   // UNICODE_TO_GBK[24826] := 16#7BB0;
   // UNICODE_TO_GBK[24827] := 16#B990;
   // UNICODE_TO_GBK[24828] := 16#7BB1;
   // UNICODE_TO_GBK[24829] := 16#CFE4;
   // UNICODE_TO_GBK[24830] := 16#7BB2;
   // UNICODE_TO_GBK[24831] := 16#B991;
   // UNICODE_TO_GBK[24832] := 16#7BB3;
   // UNICODE_TO_GBK[24833] := 16#B992;
   // UNICODE_TO_GBK[24834] := 16#7BB4;
   // UNICODE_TO_GBK[24835] := 16#F3F0;
   // UNICODE_TO_GBK[24836] := 16#7BB5;
   // UNICODE_TO_GBK[24837] := 16#B993;
   // UNICODE_TO_GBK[24838] := 16#7BB6;
   // UNICODE_TO_GBK[24839] := 16#B994;
   // UNICODE_TO_GBK[24840] := 16#7BB7;
   // UNICODE_TO_GBK[24841] := 16#B995;
   // UNICODE_TO_GBK[24842] := 16#7BB8;
   // UNICODE_TO_GBK[24843] := 16#F3E7;
   // UNICODE_TO_GBK[24844] := 16#7BB9;
   // UNICODE_TO_GBK[24845] := 16#B996;
   // UNICODE_TO_GBK[24846] := 16#7BBA;
   // UNICODE_TO_GBK[24847] := 16#B997;
   // UNICODE_TO_GBK[24848] := 16#7BBB;
   // UNICODE_TO_GBK[24849] := 16#B998;
   // UNICODE_TO_GBK[24850] := 16#7BBC;
   // UNICODE_TO_GBK[24851] := 16#B999;
   // UNICODE_TO_GBK[24852] := 16#7BBD;
   // UNICODE_TO_GBK[24853] := 16#B99A;
   // UNICODE_TO_GBK[24854] := 16#7BBE;
   // UNICODE_TO_GBK[24855] := 16#B99B;
   // UNICODE_TO_GBK[24856] := 16#7BBF;
   // UNICODE_TO_GBK[24857] := 16#B99C;
   // UNICODE_TO_GBK[24858] := 16#7BC0;
   // UNICODE_TO_GBK[24859] := 16#B99D;
   // UNICODE_TO_GBK[24860] := 16#7BC1;
   // UNICODE_TO_GBK[24861] := 16#F3F2;
   // UNICODE_TO_GBK[24862] := 16#7BC2;
   // UNICODE_TO_GBK[24863] := 16#B99E;
   // UNICODE_TO_GBK[24864] := 16#7BC3;
   // UNICODE_TO_GBK[24865] := 16#B99F;
   // UNICODE_TO_GBK[24866] := 16#7BC4;
   // UNICODE_TO_GBK[24867] := 16#B9A0;
   // UNICODE_TO_GBK[24868] := 16#7BC5;
   // UNICODE_TO_GBK[24869] := 16#BA40;
   // UNICODE_TO_GBK[24870] := 16#7BC6;
   // UNICODE_TO_GBK[24871] := 16#D7AD;
   // UNICODE_TO_GBK[24872] := 16#7BC7;
   // UNICODE_TO_GBK[24873] := 16#C6AA;
   // UNICODE_TO_GBK[24874] := 16#7BC8;
   // UNICODE_TO_GBK[24875] := 16#BA41;
   // UNICODE_TO_GBK[24876] := 16#7BC9;
   // UNICODE_TO_GBK[24877] := 16#BA42;
   // UNICODE_TO_GBK[24878] := 16#7BCA;
   // UNICODE_TO_GBK[24879] := 16#BA43;
   // UNICODE_TO_GBK[24880] := 16#7BCB;
   // UNICODE_TO_GBK[24881] := 16#BA44;
   // UNICODE_TO_GBK[24882] := 16#7BCC;
   // UNICODE_TO_GBK[24883] := 16#F3F3;
   // UNICODE_TO_GBK[24884] := 16#7BCD;
   // UNICODE_TO_GBK[24885] := 16#BA45;
   // UNICODE_TO_GBK[24886] := 16#7BCE;
   // UNICODE_TO_GBK[24887] := 16#BA46;
   // UNICODE_TO_GBK[24888] := 16#7BCF;
   // UNICODE_TO_GBK[24889] := 16#BA47;
   // UNICODE_TO_GBK[24890] := 16#7BD0;
   // UNICODE_TO_GBK[24891] := 16#BA48;
   // UNICODE_TO_GBK[24892] := 16#7BD1;
   // UNICODE_TO_GBK[24893] := 16#F3F1;
   // UNICODE_TO_GBK[24894] := 16#7BD2;
   // UNICODE_TO_GBK[24895] := 16#BA49;
   // UNICODE_TO_GBK[24896] := 16#7BD3;
   // UNICODE_TO_GBK[24897] := 16#C2A8;
   // UNICODE_TO_GBK[24898] := 16#7BD4;
   // UNICODE_TO_GBK[24899] := 16#BA4A;
   // UNICODE_TO_GBK[24900] := 16#7BD5;
   // UNICODE_TO_GBK[24901] := 16#BA4B;
   // UNICODE_TO_GBK[24902] := 16#7BD6;
   // UNICODE_TO_GBK[24903] := 16#BA4C;
   // UNICODE_TO_GBK[24904] := 16#7BD7;
   // UNICODE_TO_GBK[24905] := 16#BA4D;
   // UNICODE_TO_GBK[24906] := 16#7BD8;
   // UNICODE_TO_GBK[24907] := 16#BA4E;
   // UNICODE_TO_GBK[24908] := 16#7BD9;
   // UNICODE_TO_GBK[24909] := 16#B8DD;
   // UNICODE_TO_GBK[24910] := 16#7BDA;
   // UNICODE_TO_GBK[24911] := 16#F3F5;
   // UNICODE_TO_GBK[24912] := 16#7BDB;
   // UNICODE_TO_GBK[24913] := 16#BA4F;
   // UNICODE_TO_GBK[24914] := 16#7BDC;
   // UNICODE_TO_GBK[24915] := 16#BA50;
   // UNICODE_TO_GBK[24916] := 16#7BDD;
   // UNICODE_TO_GBK[24917] := 16#F3F4;
   // UNICODE_TO_GBK[24918] := 16#7BDE;
   // UNICODE_TO_GBK[24919] := 16#BA51;
   // UNICODE_TO_GBK[24920] := 16#7BDF;
   // UNICODE_TO_GBK[24921] := 16#BA52;
   // UNICODE_TO_GBK[24922] := 16#7BE0;
   // UNICODE_TO_GBK[24923] := 16#BA53;
   // UNICODE_TO_GBK[24924] := 16#7BE1;
   // UNICODE_TO_GBK[24925] := 16#B4DB;
   // UNICODE_TO_GBK[24926] := 16#7BE2;
   // UNICODE_TO_GBK[24927] := 16#BA54;
   // UNICODE_TO_GBK[24928] := 16#7BE3;
   // UNICODE_TO_GBK[24929] := 16#BA55;
   // UNICODE_TO_GBK[24930] := 16#7BE4;
   // UNICODE_TO_GBK[24931] := 16#BA56;
   // UNICODE_TO_GBK[24932] := 16#7BE5;
   // UNICODE_TO_GBK[24933] := 16#F3F6;
   // UNICODE_TO_GBK[24934] := 16#7BE6;
   // UNICODE_TO_GBK[24935] := 16#F3F7;
   // UNICODE_TO_GBK[24936] := 16#7BE7;
   // UNICODE_TO_GBK[24937] := 16#BA57;
   // UNICODE_TO_GBK[24938] := 16#7BE8;
   // UNICODE_TO_GBK[24939] := 16#BA58;
   // UNICODE_TO_GBK[24940] := 16#7BE9;
   // UNICODE_TO_GBK[24941] := 16#BA59;
   // UNICODE_TO_GBK[24942] := 16#7BEA;
   // UNICODE_TO_GBK[24943] := 16#F3F8;
   // UNICODE_TO_GBK[24944] := 16#7BEB;
   // UNICODE_TO_GBK[24945] := 16#BA5A;
   // UNICODE_TO_GBK[24946] := 16#7BEC;
   // UNICODE_TO_GBK[24947] := 16#BA5B;
   // UNICODE_TO_GBK[24948] := 16#7BED;
   // UNICODE_TO_GBK[24949] := 16#BA5C;
   // UNICODE_TO_GBK[24950] := 16#7BEE;
   // UNICODE_TO_GBK[24951] := 16#C0BA;
   // UNICODE_TO_GBK[24952] := 16#7BEF;
   // UNICODE_TO_GBK[24953] := 16#BA5D;
   // UNICODE_TO_GBK[24954] := 16#7BF0;
   // UNICODE_TO_GBK[24955] := 16#BA5E;
   // UNICODE_TO_GBK[24956] := 16#7BF1;
   // UNICODE_TO_GBK[24957] := 16#C0E9;
   // UNICODE_TO_GBK[24958] := 16#7BF2;
   // UNICODE_TO_GBK[24959] := 16#BA5F;
   // UNICODE_TO_GBK[24960] := 16#7BF3;
   // UNICODE_TO_GBK[24961] := 16#BA60;
   // UNICODE_TO_GBK[24962] := 16#7BF4;
   // UNICODE_TO_GBK[24963] := 16#BA61;
   // UNICODE_TO_GBK[24964] := 16#7BF5;
   // UNICODE_TO_GBK[24965] := 16#BA62;
   // UNICODE_TO_GBK[24966] := 16#7BF6;
   // UNICODE_TO_GBK[24967] := 16#BA63;
   // UNICODE_TO_GBK[24968] := 16#7BF7;
   // UNICODE_TO_GBK[24969] := 16#C5F1;
   // UNICODE_TO_GBK[24970] := 16#7BF8;
   // UNICODE_TO_GBK[24971] := 16#BA64;
   // UNICODE_TO_GBK[24972] := 16#7BF9;
   // UNICODE_TO_GBK[24973] := 16#BA65;
   // UNICODE_TO_GBK[24974] := 16#7BFA;
   // UNICODE_TO_GBK[24975] := 16#BA66;
   // UNICODE_TO_GBK[24976] := 16#7BFB;
   // UNICODE_TO_GBK[24977] := 16#BA67;
   // UNICODE_TO_GBK[24978] := 16#7BFC;
   // UNICODE_TO_GBK[24979] := 16#F3FB;
   // UNICODE_TO_GBK[24980] := 16#7BFD;
   // UNICODE_TO_GBK[24981] := 16#BA68;
   // UNICODE_TO_GBK[24982] := 16#7BFE;
   // UNICODE_TO_GBK[24983] := 16#F3FA;
   // UNICODE_TO_GBK[24984] := 16#7BFF;
   // UNICODE_TO_GBK[24985] := 16#BA69;
   // UNICODE_TO_GBK[24986] := 16#7C00;
   // UNICODE_TO_GBK[24987] := 16#BA6A;
   // UNICODE_TO_GBK[24988] := 16#7C01;
   // UNICODE_TO_GBK[24989] := 16#BA6B;
   // UNICODE_TO_GBK[24990] := 16#7C02;
   // UNICODE_TO_GBK[24991] := 16#BA6C;
   // UNICODE_TO_GBK[24992] := 16#7C03;
   // UNICODE_TO_GBK[24993] := 16#BA6D;
   // UNICODE_TO_GBK[24994] := 16#7C04;
   // UNICODE_TO_GBK[24995] := 16#BA6E;
   // UNICODE_TO_GBK[24996] := 16#7C05;
   // UNICODE_TO_GBK[24997] := 16#BA6F;
   // UNICODE_TO_GBK[24998] := 16#7C06;
   // UNICODE_TO_GBK[24999] := 16#BA70;
   // UNICODE_TO_GBK[25000] := 16#7C07;
   // UNICODE_TO_GBK[25001] := 16#B4D8;
   // UNICODE_TO_GBK[25002] := 16#7C08;
   // UNICODE_TO_GBK[25003] := 16#BA71;
   // UNICODE_TO_GBK[25004] := 16#7C09;
   // UNICODE_TO_GBK[25005] := 16#BA72;
   // UNICODE_TO_GBK[25006] := 16#7C0A;
   // UNICODE_TO_GBK[25007] := 16#BA73;
   // UNICODE_TO_GBK[25008] := 16#7C0B;
   // UNICODE_TO_GBK[25009] := 16#F3FE;
   // UNICODE_TO_GBK[25010] := 16#7C0C;
   // UNICODE_TO_GBK[25011] := 16#F3F9;
   // UNICODE_TO_GBK[25012] := 16#7C0D;
   // UNICODE_TO_GBK[25013] := 16#BA74;
   // UNICODE_TO_GBK[25014] := 16#7C0E;
   // UNICODE_TO_GBK[25015] := 16#BA75;
   // UNICODE_TO_GBK[25016] := 16#7C0F;
   // UNICODE_TO_GBK[25017] := 16#F3FC;
   // UNICODE_TO_GBK[25018] := 16#7C10;
   // UNICODE_TO_GBK[25019] := 16#BA76;
   // UNICODE_TO_GBK[25020] := 16#7C11;
   // UNICODE_TO_GBK[25021] := 16#BA77;
   // UNICODE_TO_GBK[25022] := 16#7C12;
   // UNICODE_TO_GBK[25023] := 16#BA78;
   // UNICODE_TO_GBK[25024] := 16#7C13;
   // UNICODE_TO_GBK[25025] := 16#BA79;
   // UNICODE_TO_GBK[25026] := 16#7C14;
   // UNICODE_TO_GBK[25027] := 16#BA7A;
   // UNICODE_TO_GBK[25028] := 16#7C15;
   // UNICODE_TO_GBK[25029] := 16#BA7B;
   // UNICODE_TO_GBK[25030] := 16#7C16;
   // UNICODE_TO_GBK[25031] := 16#F3FD;
   // UNICODE_TO_GBK[25032] := 16#7C17;
   // UNICODE_TO_GBK[25033] := 16#BA7C;
   // UNICODE_TO_GBK[25034] := 16#7C18;
   // UNICODE_TO_GBK[25035] := 16#BA7D;
   // UNICODE_TO_GBK[25036] := 16#7C19;
   // UNICODE_TO_GBK[25037] := 16#BA7E;
   // UNICODE_TO_GBK[25038] := 16#7C1A;
   // UNICODE_TO_GBK[25039] := 16#BA80;
   // UNICODE_TO_GBK[25040] := 16#7C1B;
   // UNICODE_TO_GBK[25041] := 16#BA81;
   // UNICODE_TO_GBK[25042] := 16#7C1C;
   // UNICODE_TO_GBK[25043] := 16#BA82;
   // UNICODE_TO_GBK[25044] := 16#7C1D;
   // UNICODE_TO_GBK[25045] := 16#BA83;
   // UNICODE_TO_GBK[25046] := 16#7C1E;
   // UNICODE_TO_GBK[25047] := 16#BA84;
   // UNICODE_TO_GBK[25048] := 16#7C1F;
   // UNICODE_TO_GBK[25049] := 16#F4A1;
   // UNICODE_TO_GBK[25050] := 16#7C20;
   // UNICODE_TO_GBK[25051] := 16#BA85;
   // UNICODE_TO_GBK[25052] := 16#7C21;
   // UNICODE_TO_GBK[25053] := 16#BA86;
   // UNICODE_TO_GBK[25054] := 16#7C22;
   // UNICODE_TO_GBK[25055] := 16#BA87;
   // UNICODE_TO_GBK[25056] := 16#7C23;
   // UNICODE_TO_GBK[25057] := 16#BA88;
   // UNICODE_TO_GBK[25058] := 16#7C24;
   // UNICODE_TO_GBK[25059] := 16#BA89;
   // UNICODE_TO_GBK[25060] := 16#7C25;
   // UNICODE_TO_GBK[25061] := 16#BA8A;
   // UNICODE_TO_GBK[25062] := 16#7C26;
   // UNICODE_TO_GBK[25063] := 16#F4A3;
   // UNICODE_TO_GBK[25064] := 16#7C27;
   // UNICODE_TO_GBK[25065] := 16#BBC9;
   // UNICODE_TO_GBK[25066] := 16#7C28;
   // UNICODE_TO_GBK[25067] := 16#BA8B;
   // UNICODE_TO_GBK[25068] := 16#7C29;
   // UNICODE_TO_GBK[25069] := 16#BA8C;
   // UNICODE_TO_GBK[25070] := 16#7C2A;
   // UNICODE_TO_GBK[25071] := 16#F4A2;
   // UNICODE_TO_GBK[25072] := 16#7C2B;
   // UNICODE_TO_GBK[25073] := 16#BA8D;
   // UNICODE_TO_GBK[25074] := 16#7C2C;
   // UNICODE_TO_GBK[25075] := 16#BA8E;
   // UNICODE_TO_GBK[25076] := 16#7C2D;
   // UNICODE_TO_GBK[25077] := 16#BA8F;
   // UNICODE_TO_GBK[25078] := 16#7C2E;
   // UNICODE_TO_GBK[25079] := 16#BA90;
   // UNICODE_TO_GBK[25080] := 16#7C2F;
   // UNICODE_TO_GBK[25081] := 16#BA91;
   // UNICODE_TO_GBK[25082] := 16#7C30;
   // UNICODE_TO_GBK[25083] := 16#BA92;
   // UNICODE_TO_GBK[25084] := 16#7C31;
   // UNICODE_TO_GBK[25085] := 16#BA93;
   // UNICODE_TO_GBK[25086] := 16#7C32;
   // UNICODE_TO_GBK[25087] := 16#BA94;
   // UNICODE_TO_GBK[25088] := 16#7C33;
   // UNICODE_TO_GBK[25089] := 16#BA95;
   // UNICODE_TO_GBK[25090] := 16#7C34;
   // UNICODE_TO_GBK[25091] := 16#BA96;
   // UNICODE_TO_GBK[25092] := 16#7C35;
   // UNICODE_TO_GBK[25093] := 16#BA97;
   // UNICODE_TO_GBK[25094] := 16#7C36;
   // UNICODE_TO_GBK[25095] := 16#BA98;
   // UNICODE_TO_GBK[25096] := 16#7C37;
   // UNICODE_TO_GBK[25097] := 16#BA99;
   // UNICODE_TO_GBK[25098] := 16#7C38;
   // UNICODE_TO_GBK[25099] := 16#F4A4;
   // UNICODE_TO_GBK[25100] := 16#7C39;
   // UNICODE_TO_GBK[25101] := 16#BA9A;
   // UNICODE_TO_GBK[25102] := 16#7C3A;
   // UNICODE_TO_GBK[25103] := 16#BA9B;
   // UNICODE_TO_GBK[25104] := 16#7C3B;
   // UNICODE_TO_GBK[25105] := 16#BA9C;
   // UNICODE_TO_GBK[25106] := 16#7C3C;
   // UNICODE_TO_GBK[25107] := 16#BA9D;
   // UNICODE_TO_GBK[25108] := 16#7C3D;
   // UNICODE_TO_GBK[25109] := 16#BA9E;
   // UNICODE_TO_GBK[25110] := 16#7C3E;
   // UNICODE_TO_GBK[25111] := 16#BA9F;
   // UNICODE_TO_GBK[25112] := 16#7C3F;
   // UNICODE_TO_GBK[25113] := 16#B2BE;
   // UNICODE_TO_GBK[25114] := 16#7C40;
   // UNICODE_TO_GBK[25115] := 16#F4A6;
   // UNICODE_TO_GBK[25116] := 16#7C41;
   // UNICODE_TO_GBK[25117] := 16#F4A5;
   // UNICODE_TO_GBK[25118] := 16#7C42;
   // UNICODE_TO_GBK[25119] := 16#BAA0;
   // UNICODE_TO_GBK[25120] := 16#7C43;
   // UNICODE_TO_GBK[25121] := 16#BB40;
   // UNICODE_TO_GBK[25122] := 16#7C44;
   // UNICODE_TO_GBK[25123] := 16#BB41;
   // UNICODE_TO_GBK[25124] := 16#7C45;
   // UNICODE_TO_GBK[25125] := 16#BB42;
   // UNICODE_TO_GBK[25126] := 16#7C46;
   // UNICODE_TO_GBK[25127] := 16#BB43;
   // UNICODE_TO_GBK[25128] := 16#7C47;
   // UNICODE_TO_GBK[25129] := 16#BB44;
   // UNICODE_TO_GBK[25130] := 16#7C48;
   // UNICODE_TO_GBK[25131] := 16#BB45;
   // UNICODE_TO_GBK[25132] := 16#7C49;
   // UNICODE_TO_GBK[25133] := 16#BB46;
   // UNICODE_TO_GBK[25134] := 16#7C4A;
   // UNICODE_TO_GBK[25135] := 16#BB47;
   // UNICODE_TO_GBK[25136] := 16#7C4B;
   // UNICODE_TO_GBK[25137] := 16#BB48;
   // UNICODE_TO_GBK[25138] := 16#7C4C;
   // UNICODE_TO_GBK[25139] := 16#BB49;
   // UNICODE_TO_GBK[25140] := 16#7C4D;
   // UNICODE_TO_GBK[25141] := 16#BCAE;
   // UNICODE_TO_GBK[25142] := 16#7C4E;
   // UNICODE_TO_GBK[25143] := 16#BB4A;
   // UNICODE_TO_GBK[25144] := 16#7C4F;
   // UNICODE_TO_GBK[25145] := 16#BB4B;
   // UNICODE_TO_GBK[25146] := 16#7C50;
   // UNICODE_TO_GBK[25147] := 16#BB4C;
   // UNICODE_TO_GBK[25148] := 16#7C51;
   // UNICODE_TO_GBK[25149] := 16#BB4D;
   // UNICODE_TO_GBK[25150] := 16#7C52;
   // UNICODE_TO_GBK[25151] := 16#BB4E;
   // UNICODE_TO_GBK[25152] := 16#7C53;
   // UNICODE_TO_GBK[25153] := 16#BB4F;
   // UNICODE_TO_GBK[25154] := 16#7C54;
   // UNICODE_TO_GBK[25155] := 16#BB50;
   // UNICODE_TO_GBK[25156] := 16#7C55;
   // UNICODE_TO_GBK[25157] := 16#BB51;
   // UNICODE_TO_GBK[25158] := 16#7C56;
   // UNICODE_TO_GBK[25159] := 16#BB52;
   // UNICODE_TO_GBK[25160] := 16#7C57;
   // UNICODE_TO_GBK[25161] := 16#BB53;
   // UNICODE_TO_GBK[25162] := 16#7C58;
   // UNICODE_TO_GBK[25163] := 16#BB54;
   // UNICODE_TO_GBK[25164] := 16#7C59;
   // UNICODE_TO_GBK[25165] := 16#BB55;
   // UNICODE_TO_GBK[25166] := 16#7C5A;
   // UNICODE_TO_GBK[25167] := 16#BB56;
   // UNICODE_TO_GBK[25168] := 16#7C5B;
   // UNICODE_TO_GBK[25169] := 16#BB57;
   // UNICODE_TO_GBK[25170] := 16#7C5C;
   // UNICODE_TO_GBK[25171] := 16#BB58;
   // UNICODE_TO_GBK[25172] := 16#7C5D;
   // UNICODE_TO_GBK[25173] := 16#BB59;
   // UNICODE_TO_GBK[25174] := 16#7C5E;
   // UNICODE_TO_GBK[25175] := 16#BB5A;
   // UNICODE_TO_GBK[25176] := 16#7C5F;
   // UNICODE_TO_GBK[25177] := 16#BB5B;
   // UNICODE_TO_GBK[25178] := 16#7C60;
   // UNICODE_TO_GBK[25179] := 16#BB5C;
   // UNICODE_TO_GBK[25180] := 16#7C61;
   // UNICODE_TO_GBK[25181] := 16#BB5D;
   // UNICODE_TO_GBK[25182] := 16#7C62;
   // UNICODE_TO_GBK[25183] := 16#BB5E;
   // UNICODE_TO_GBK[25184] := 16#7C63;
   // UNICODE_TO_GBK[25185] := 16#BB5F;
   // UNICODE_TO_GBK[25186] := 16#7C64;
   // UNICODE_TO_GBK[25187] := 16#BB60;
   // UNICODE_TO_GBK[25188] := 16#7C65;
   // UNICODE_TO_GBK[25189] := 16#BB61;
   // UNICODE_TO_GBK[25190] := 16#7C66;
   // UNICODE_TO_GBK[25191] := 16#BB62;
   // UNICODE_TO_GBK[25192] := 16#7C67;
   // UNICODE_TO_GBK[25193] := 16#BB63;
   // UNICODE_TO_GBK[25194] := 16#7C68;
   // UNICODE_TO_GBK[25195] := 16#BB64;
   // UNICODE_TO_GBK[25196] := 16#7C69;
   // UNICODE_TO_GBK[25197] := 16#BB65;
   // UNICODE_TO_GBK[25198] := 16#7C6A;
   // UNICODE_TO_GBK[25199] := 16#BB66;
   // UNICODE_TO_GBK[25200] := 16#7C6B;
   // UNICODE_TO_GBK[25201] := 16#BB67;
   // UNICODE_TO_GBK[25202] := 16#7C6C;
   // UNICODE_TO_GBK[25203] := 16#BB68;
   // UNICODE_TO_GBK[25204] := 16#7C6D;
   // UNICODE_TO_GBK[25205] := 16#BB69;
   // UNICODE_TO_GBK[25206] := 16#7C6E;
   // UNICODE_TO_GBK[25207] := 16#BB6A;
   // UNICODE_TO_GBK[25208] := 16#7C6F;
   // UNICODE_TO_GBK[25209] := 16#BB6B;
   // UNICODE_TO_GBK[25210] := 16#7C70;
   // UNICODE_TO_GBK[25211] := 16#BB6C;
   // UNICODE_TO_GBK[25212] := 16#7C71;
   // UNICODE_TO_GBK[25213] := 16#BB6D;
   // UNICODE_TO_GBK[25214] := 16#7C72;
   // UNICODE_TO_GBK[25215] := 16#BB6E;
   // UNICODE_TO_GBK[25216] := 16#7C73;
   // UNICODE_TO_GBK[25217] := 16#C3D7;
   // UNICODE_TO_GBK[25218] := 16#7C74;
   // UNICODE_TO_GBK[25219] := 16#D9E1;
   // UNICODE_TO_GBK[25220] := 16#7C75;
   // UNICODE_TO_GBK[25221] := 16#BB6F;
   // UNICODE_TO_GBK[25222] := 16#7C76;
   // UNICODE_TO_GBK[25223] := 16#BB70;
   // UNICODE_TO_GBK[25224] := 16#7C77;
   // UNICODE_TO_GBK[25225] := 16#BB71;
   // UNICODE_TO_GBK[25226] := 16#7C78;
   // UNICODE_TO_GBK[25227] := 16#BB72;
   // UNICODE_TO_GBK[25228] := 16#7C79;
   // UNICODE_TO_GBK[25229] := 16#BB73;
   // UNICODE_TO_GBK[25230] := 16#7C7A;
   // UNICODE_TO_GBK[25231] := 16#BB74;
   // UNICODE_TO_GBK[25232] := 16#7C7B;
   // UNICODE_TO_GBK[25233] := 16#C0E0;
   // UNICODE_TO_GBK[25234] := 16#7C7C;
   // UNICODE_TO_GBK[25235] := 16#F4CC;
   // UNICODE_TO_GBK[25236] := 16#7C7D;
   // UNICODE_TO_GBK[25237] := 16#D7D1;
   // UNICODE_TO_GBK[25238] := 16#7C7E;
   // UNICODE_TO_GBK[25239] := 16#BB75;
   // UNICODE_TO_GBK[25240] := 16#7C7F;
   // UNICODE_TO_GBK[25241] := 16#BB76;
   // UNICODE_TO_GBK[25242] := 16#7C80;
   // UNICODE_TO_GBK[25243] := 16#BB77;
   // UNICODE_TO_GBK[25244] := 16#7C81;
   // UNICODE_TO_GBK[25245] := 16#BB78;
   // UNICODE_TO_GBK[25246] := 16#7C82;
   // UNICODE_TO_GBK[25247] := 16#BB79;
   // UNICODE_TO_GBK[25248] := 16#7C83;
   // UNICODE_TO_GBK[25249] := 16#BB7A;
   // UNICODE_TO_GBK[25250] := 16#7C84;
   // UNICODE_TO_GBK[25251] := 16#BB7B;
   // UNICODE_TO_GBK[25252] := 16#7C85;
   // UNICODE_TO_GBK[25253] := 16#BB7C;
   // UNICODE_TO_GBK[25254] := 16#7C86;
   // UNICODE_TO_GBK[25255] := 16#BB7D;
   // UNICODE_TO_GBK[25256] := 16#7C87;
   // UNICODE_TO_GBK[25257] := 16#BB7E;
   // UNICODE_TO_GBK[25258] := 16#7C88;
   // UNICODE_TO_GBK[25259] := 16#BB80;
   // UNICODE_TO_GBK[25260] := 16#7C89;
   // UNICODE_TO_GBK[25261] := 16#B7DB;
   // UNICODE_TO_GBK[25262] := 16#7C8A;
   // UNICODE_TO_GBK[25263] := 16#BB81;
   // UNICODE_TO_GBK[25264] := 16#7C8B;
   // UNICODE_TO_GBK[25265] := 16#BB82;
   // UNICODE_TO_GBK[25266] := 16#7C8C;
   // UNICODE_TO_GBK[25267] := 16#BB83;
   // UNICODE_TO_GBK[25268] := 16#7C8D;
   // UNICODE_TO_GBK[25269] := 16#BB84;
   // UNICODE_TO_GBK[25270] := 16#7C8E;
   // UNICODE_TO_GBK[25271] := 16#BB85;
   // UNICODE_TO_GBK[25272] := 16#7C8F;
   // UNICODE_TO_GBK[25273] := 16#BB86;
   // UNICODE_TO_GBK[25274] := 16#7C90;
   // UNICODE_TO_GBK[25275] := 16#BB87;
   // UNICODE_TO_GBK[25276] := 16#7C91;
   // UNICODE_TO_GBK[25277] := 16#F4CE;
   // UNICODE_TO_GBK[25278] := 16#7C92;
   // UNICODE_TO_GBK[25279] := 16#C1A3;
   // UNICODE_TO_GBK[25280] := 16#7C93;
   // UNICODE_TO_GBK[25281] := 16#BB88;
   // UNICODE_TO_GBK[25282] := 16#7C94;
   // UNICODE_TO_GBK[25283] := 16#BB89;
   // UNICODE_TO_GBK[25284] := 16#7C95;
   // UNICODE_TO_GBK[25285] := 16#C6C9;
   // UNICODE_TO_GBK[25286] := 16#7C96;
   // UNICODE_TO_GBK[25287] := 16#BB8A;
   // UNICODE_TO_GBK[25288] := 16#7C97;
   // UNICODE_TO_GBK[25289] := 16#B4D6;
   // UNICODE_TO_GBK[25290] := 16#7C98;
   // UNICODE_TO_GBK[25291] := 16#D5B3;
   // UNICODE_TO_GBK[25292] := 16#7C99;
   // UNICODE_TO_GBK[25293] := 16#BB8B;
   // UNICODE_TO_GBK[25294] := 16#7C9A;
   // UNICODE_TO_GBK[25295] := 16#BB8C;
   // UNICODE_TO_GBK[25296] := 16#7C9B;
   // UNICODE_TO_GBK[25297] := 16#BB8D;
   // UNICODE_TO_GBK[25298] := 16#7C9C;
   // UNICODE_TO_GBK[25299] := 16#F4D0;
   // UNICODE_TO_GBK[25300] := 16#7C9D;
   // UNICODE_TO_GBK[25301] := 16#F4CF;
   // UNICODE_TO_GBK[25302] := 16#7C9E;
   // UNICODE_TO_GBK[25303] := 16#F4D1;
   // UNICODE_TO_GBK[25304] := 16#7C9F;
   // UNICODE_TO_GBK[25305] := 16#CBDA;
   // UNICODE_TO_GBK[25306] := 16#7CA0;
   // UNICODE_TO_GBK[25307] := 16#BB8E;
   // UNICODE_TO_GBK[25308] := 16#7CA1;
   // UNICODE_TO_GBK[25309] := 16#BB8F;
   // UNICODE_TO_GBK[25310] := 16#7CA2;
   // UNICODE_TO_GBK[25311] := 16#F4D2;
   // UNICODE_TO_GBK[25312] := 16#7CA3;
   // UNICODE_TO_GBK[25313] := 16#BB90;
   // UNICODE_TO_GBK[25314] := 16#7CA4;
   // UNICODE_TO_GBK[25315] := 16#D4C1;
   // UNICODE_TO_GBK[25316] := 16#7CA5;
   // UNICODE_TO_GBK[25317] := 16#D6E0;
   // UNICODE_TO_GBK[25318] := 16#7CA6;
   // UNICODE_TO_GBK[25319] := 16#BB91;
   // UNICODE_TO_GBK[25320] := 16#7CA7;
   // UNICODE_TO_GBK[25321] := 16#BB92;
   // UNICODE_TO_GBK[25322] := 16#7CA8;
   // UNICODE_TO_GBK[25323] := 16#BB93;
   // UNICODE_TO_GBK[25324] := 16#7CA9;
   // UNICODE_TO_GBK[25325] := 16#BB94;
   // UNICODE_TO_GBK[25326] := 16#7CAA;
   // UNICODE_TO_GBK[25327] := 16#B7E0;
   // UNICODE_TO_GBK[25328] := 16#7CAB;
   // UNICODE_TO_GBK[25329] := 16#BB95;
   // UNICODE_TO_GBK[25330] := 16#7CAC;
   // UNICODE_TO_GBK[25331] := 16#BB96;
   // UNICODE_TO_GBK[25332] := 16#7CAD;
   // UNICODE_TO_GBK[25333] := 16#BB97;
   // UNICODE_TO_GBK[25334] := 16#7CAE;
   // UNICODE_TO_GBK[25335] := 16#C1B8;
   // UNICODE_TO_GBK[25336] := 16#7CAF;
   // UNICODE_TO_GBK[25337] := 16#BB98;
   // UNICODE_TO_GBK[25338] := 16#7CB0;
   // UNICODE_TO_GBK[25339] := 16#BB99;
   // UNICODE_TO_GBK[25340] := 16#7CB1;
   // UNICODE_TO_GBK[25341] := 16#C1BB;
   // UNICODE_TO_GBK[25342] := 16#7CB2;
   // UNICODE_TO_GBK[25343] := 16#F4D3;
   // UNICODE_TO_GBK[25344] := 16#7CB3;
   // UNICODE_TO_GBK[25345] := 16#BEAC;
   // UNICODE_TO_GBK[25346] := 16#7CB4;
   // UNICODE_TO_GBK[25347] := 16#BB9A;
   // UNICODE_TO_GBK[25348] := 16#7CB5;
   // UNICODE_TO_GBK[25349] := 16#BB9B;
   // UNICODE_TO_GBK[25350] := 16#7CB6;
   // UNICODE_TO_GBK[25351] := 16#BB9C;
   // UNICODE_TO_GBK[25352] := 16#7CB7;
   // UNICODE_TO_GBK[25353] := 16#BB9D;
   // UNICODE_TO_GBK[25354] := 16#7CB8;
   // UNICODE_TO_GBK[25355] := 16#BB9E;
   // UNICODE_TO_GBK[25356] := 16#7CB9;
   // UNICODE_TO_GBK[25357] := 16#B4E2;
   // UNICODE_TO_GBK[25358] := 16#7CBA;
   // UNICODE_TO_GBK[25359] := 16#BB9F;
   // UNICODE_TO_GBK[25360] := 16#7CBB;
   // UNICODE_TO_GBK[25361] := 16#BBA0;
   // UNICODE_TO_GBK[25362] := 16#7CBC;
   // UNICODE_TO_GBK[25363] := 16#F4D4;
   // UNICODE_TO_GBK[25364] := 16#7CBD;
   // UNICODE_TO_GBK[25365] := 16#F4D5;
   // UNICODE_TO_GBK[25366] := 16#7CBE;
   // UNICODE_TO_GBK[25367] := 16#BEAB;
   // UNICODE_TO_GBK[25368] := 16#7CBF;
   // UNICODE_TO_GBK[25369] := 16#BC40;
   // UNICODE_TO_GBK[25370] := 16#7CC0;
   // UNICODE_TO_GBK[25371] := 16#BC41;
   // UNICODE_TO_GBK[25372] := 16#7CC1;
   // UNICODE_TO_GBK[25373] := 16#F4D6;
   // UNICODE_TO_GBK[25374] := 16#7CC2;
   // UNICODE_TO_GBK[25375] := 16#BC42;
   // UNICODE_TO_GBK[25376] := 16#7CC3;
   // UNICODE_TO_GBK[25377] := 16#BC43;
   // UNICODE_TO_GBK[25378] := 16#7CC4;
   // UNICODE_TO_GBK[25379] := 16#BC44;
   // UNICODE_TO_GBK[25380] := 16#7CC5;
   // UNICODE_TO_GBK[25381] := 16#F4DB;
   // UNICODE_TO_GBK[25382] := 16#7CC6;
   // UNICODE_TO_GBK[25383] := 16#BC45;
   // UNICODE_TO_GBK[25384] := 16#7CC7;
   // UNICODE_TO_GBK[25385] := 16#F4D7;
   // UNICODE_TO_GBK[25386] := 16#7CC8;
   // UNICODE_TO_GBK[25387] := 16#F4DA;
   // UNICODE_TO_GBK[25388] := 16#7CC9;
   // UNICODE_TO_GBK[25389] := 16#BC46;
   // UNICODE_TO_GBK[25390] := 16#7CCA;
   // UNICODE_TO_GBK[25391] := 16#BAFD;
   // UNICODE_TO_GBK[25392] := 16#7CCB;
   // UNICODE_TO_GBK[25393] := 16#BC47;
   // UNICODE_TO_GBK[25394] := 16#7CCC;
   // UNICODE_TO_GBK[25395] := 16#F4D8;
   // UNICODE_TO_GBK[25396] := 16#7CCD;
   // UNICODE_TO_GBK[25397] := 16#F4D9;
   // UNICODE_TO_GBK[25398] := 16#7CCE;
   // UNICODE_TO_GBK[25399] := 16#BC48;
   // UNICODE_TO_GBK[25400] := 16#7CCF;
   // UNICODE_TO_GBK[25401] := 16#BC49;
   // UNICODE_TO_GBK[25402] := 16#7CD0;
   // UNICODE_TO_GBK[25403] := 16#BC4A;
   // UNICODE_TO_GBK[25404] := 16#7CD1;
   // UNICODE_TO_GBK[25405] := 16#BC4B;
   // UNICODE_TO_GBK[25406] := 16#7CD2;
   // UNICODE_TO_GBK[25407] := 16#BC4C;
   // UNICODE_TO_GBK[25408] := 16#7CD3;
   // UNICODE_TO_GBK[25409] := 16#BC4D;
   // UNICODE_TO_GBK[25410] := 16#7CD4;
   // UNICODE_TO_GBK[25411] := 16#BC4E;
   // UNICODE_TO_GBK[25412] := 16#7CD5;
   // UNICODE_TO_GBK[25413] := 16#B8E2;
   // UNICODE_TO_GBK[25414] := 16#7CD6;
   // UNICODE_TO_GBK[25415] := 16#CCC7;
   // UNICODE_TO_GBK[25416] := 16#7CD7;
   // UNICODE_TO_GBK[25417] := 16#F4DC;
   // UNICODE_TO_GBK[25418] := 16#7CD8;
   // UNICODE_TO_GBK[25419] := 16#BC4F;
   // UNICODE_TO_GBK[25420] := 16#7CD9;
   // UNICODE_TO_GBK[25421] := 16#B2DA;
   // UNICODE_TO_GBK[25422] := 16#7CDA;
   // UNICODE_TO_GBK[25423] := 16#BC50;
   // UNICODE_TO_GBK[25424] := 16#7CDB;
   // UNICODE_TO_GBK[25425] := 16#BC51;
   // UNICODE_TO_GBK[25426] := 16#7CDC;
   // UNICODE_TO_GBK[25427] := 16#C3D3;
   // UNICODE_TO_GBK[25428] := 16#7CDD;
   // UNICODE_TO_GBK[25429] := 16#BC52;
   // UNICODE_TO_GBK[25430] := 16#7CDE;
   // UNICODE_TO_GBK[25431] := 16#BC53;
   // UNICODE_TO_GBK[25432] := 16#7CDF;
   // UNICODE_TO_GBK[25433] := 16#D4E3;
   // UNICODE_TO_GBK[25434] := 16#7CE0;
   // UNICODE_TO_GBK[25435] := 16#BFB7;
   // UNICODE_TO_GBK[25436] := 16#7CE1;
   // UNICODE_TO_GBK[25437] := 16#BC54;
   // UNICODE_TO_GBK[25438] := 16#7CE2;
   // UNICODE_TO_GBK[25439] := 16#BC55;
   // UNICODE_TO_GBK[25440] := 16#7CE3;
   // UNICODE_TO_GBK[25441] := 16#BC56;
   // UNICODE_TO_GBK[25442] := 16#7CE4;
   // UNICODE_TO_GBK[25443] := 16#BC57;
   // UNICODE_TO_GBK[25444] := 16#7CE5;
   // UNICODE_TO_GBK[25445] := 16#BC58;
   // UNICODE_TO_GBK[25446] := 16#7CE6;
   // UNICODE_TO_GBK[25447] := 16#BC59;
   // UNICODE_TO_GBK[25448] := 16#7CE7;
   // UNICODE_TO_GBK[25449] := 16#BC5A;
   // UNICODE_TO_GBK[25450] := 16#7CE8;
   // UNICODE_TO_GBK[25451] := 16#F4DD;
   // UNICODE_TO_GBK[25452] := 16#7CE9;
   // UNICODE_TO_GBK[25453] := 16#BC5B;
   // UNICODE_TO_GBK[25454] := 16#7CEA;
   // UNICODE_TO_GBK[25455] := 16#BC5C;
   // UNICODE_TO_GBK[25456] := 16#7CEB;
   // UNICODE_TO_GBK[25457] := 16#BC5D;
   // UNICODE_TO_GBK[25458] := 16#7CEC;
   // UNICODE_TO_GBK[25459] := 16#BC5E;
   // UNICODE_TO_GBK[25460] := 16#7CED;
   // UNICODE_TO_GBK[25461] := 16#BC5F;
   // UNICODE_TO_GBK[25462] := 16#7CEE;
   // UNICODE_TO_GBK[25463] := 16#BC60;
   // UNICODE_TO_GBK[25464] := 16#7CEF;
   // UNICODE_TO_GBK[25465] := 16#C5B4;
   // UNICODE_TO_GBK[25466] := 16#7CF0;
   // UNICODE_TO_GBK[25467] := 16#BC61;
   // UNICODE_TO_GBK[25468] := 16#7CF1;
   // UNICODE_TO_GBK[25469] := 16#BC62;
   // UNICODE_TO_GBK[25470] := 16#7CF2;
   // UNICODE_TO_GBK[25471] := 16#BC63;
   // UNICODE_TO_GBK[25472] := 16#7CF3;
   // UNICODE_TO_GBK[25473] := 16#BC64;
   // UNICODE_TO_GBK[25474] := 16#7CF4;
   // UNICODE_TO_GBK[25475] := 16#BC65;
   // UNICODE_TO_GBK[25476] := 16#7CF5;
   // UNICODE_TO_GBK[25477] := 16#BC66;
   // UNICODE_TO_GBK[25478] := 16#7CF6;
   // UNICODE_TO_GBK[25479] := 16#BC67;
   // UNICODE_TO_GBK[25480] := 16#7CF7;
   // UNICODE_TO_GBK[25481] := 16#BC68;
   // UNICODE_TO_GBK[25482] := 16#7CF8;
   // UNICODE_TO_GBK[25483] := 16#F4E9;
   // UNICODE_TO_GBK[25484] := 16#7CF9;
   // UNICODE_TO_GBK[25485] := 16#BC69;
   // UNICODE_TO_GBK[25486] := 16#7CFA;
   // UNICODE_TO_GBK[25487] := 16#BC6A;
   // UNICODE_TO_GBK[25488] := 16#7CFB;
   // UNICODE_TO_GBK[25489] := 16#CFB5;
   // UNICODE_TO_GBK[25490] := 16#7CFC;
   // UNICODE_TO_GBK[25491] := 16#BC6B;
   // UNICODE_TO_GBK[25492] := 16#7CFD;
   // UNICODE_TO_GBK[25493] := 16#BC6C;
   // UNICODE_TO_GBK[25494] := 16#7CFE;
   // UNICODE_TO_GBK[25495] := 16#BC6D;
   // UNICODE_TO_GBK[25496] := 16#7CFF;
   // UNICODE_TO_GBK[25497] := 16#BC6E;
   // UNICODE_TO_GBK[25498] := 16#7D00;
   // UNICODE_TO_GBK[25499] := 16#BC6F;
   // UNICODE_TO_GBK[25500] := 16#7D01;
   // UNICODE_TO_GBK[25501] := 16#BC70;
   // UNICODE_TO_GBK[25502] := 16#7D02;
   // UNICODE_TO_GBK[25503] := 16#BC71;
   // UNICODE_TO_GBK[25504] := 16#7D03;
   // UNICODE_TO_GBK[25505] := 16#BC72;
   // UNICODE_TO_GBK[25506] := 16#7D04;
   // UNICODE_TO_GBK[25507] := 16#BC73;
   // UNICODE_TO_GBK[25508] := 16#7D05;
   // UNICODE_TO_GBK[25509] := 16#BC74;
   // UNICODE_TO_GBK[25510] := 16#7D06;
   // UNICODE_TO_GBK[25511] := 16#BC75;
   // UNICODE_TO_GBK[25512] := 16#7D07;
   // UNICODE_TO_GBK[25513] := 16#BC76;
   // UNICODE_TO_GBK[25514] := 16#7D08;
   // UNICODE_TO_GBK[25515] := 16#BC77;
   // UNICODE_TO_GBK[25516] := 16#7D09;
   // UNICODE_TO_GBK[25517] := 16#BC78;
   // UNICODE_TO_GBK[25518] := 16#7D0A;
   // UNICODE_TO_GBK[25519] := 16#CEC9;
   // UNICODE_TO_GBK[25520] := 16#7D0B;
   // UNICODE_TO_GBK[25521] := 16#BC79;
   // UNICODE_TO_GBK[25522] := 16#7D0C;
   // UNICODE_TO_GBK[25523] := 16#BC7A;
   // UNICODE_TO_GBK[25524] := 16#7D0D;
   // UNICODE_TO_GBK[25525] := 16#BC7B;
   // UNICODE_TO_GBK[25526] := 16#7D0E;
   // UNICODE_TO_GBK[25527] := 16#BC7C;
   // UNICODE_TO_GBK[25528] := 16#7D0F;
   // UNICODE_TO_GBK[25529] := 16#BC7D;
   // UNICODE_TO_GBK[25530] := 16#7D10;
   // UNICODE_TO_GBK[25531] := 16#BC7E;
   // UNICODE_TO_GBK[25532] := 16#7D11;
   // UNICODE_TO_GBK[25533] := 16#BC80;
   // UNICODE_TO_GBK[25534] := 16#7D12;
   // UNICODE_TO_GBK[25535] := 16#BC81;
   // UNICODE_TO_GBK[25536] := 16#7D13;
   // UNICODE_TO_GBK[25537] := 16#BC82;
   // UNICODE_TO_GBK[25538] := 16#7D14;
   // UNICODE_TO_GBK[25539] := 16#BC83;
   // UNICODE_TO_GBK[25540] := 16#7D15;
   // UNICODE_TO_GBK[25541] := 16#BC84;
   // UNICODE_TO_GBK[25542] := 16#7D16;
   // UNICODE_TO_GBK[25543] := 16#BC85;
   // UNICODE_TO_GBK[25544] := 16#7D17;
   // UNICODE_TO_GBK[25545] := 16#BC86;
   // UNICODE_TO_GBK[25546] := 16#7D18;
   // UNICODE_TO_GBK[25547] := 16#BC87;
   // UNICODE_TO_GBK[25548] := 16#7D19;
   // UNICODE_TO_GBK[25549] := 16#BC88;
   // UNICODE_TO_GBK[25550] := 16#7D1A;
   // UNICODE_TO_GBK[25551] := 16#BC89;
   // UNICODE_TO_GBK[25552] := 16#7D1B;
   // UNICODE_TO_GBK[25553] := 16#BC8A;
   // UNICODE_TO_GBK[25554] := 16#7D1C;
   // UNICODE_TO_GBK[25555] := 16#BC8B;
   // UNICODE_TO_GBK[25556] := 16#7D1D;
   // UNICODE_TO_GBK[25557] := 16#BC8C;
   // UNICODE_TO_GBK[25558] := 16#7D1E;
   // UNICODE_TO_GBK[25559] := 16#BC8D;
   // UNICODE_TO_GBK[25560] := 16#7D1F;
   // UNICODE_TO_GBK[25561] := 16#BC8E;
   // UNICODE_TO_GBK[25562] := 16#7D20;
   // UNICODE_TO_GBK[25563] := 16#CBD8;
   // UNICODE_TO_GBK[25564] := 16#7D21;
   // UNICODE_TO_GBK[25565] := 16#BC8F;
   // UNICODE_TO_GBK[25566] := 16#7D22;
   // UNICODE_TO_GBK[25567] := 16#CBF7;
   // UNICODE_TO_GBK[25568] := 16#7D23;
   // UNICODE_TO_GBK[25569] := 16#BC90;
   // UNICODE_TO_GBK[25570] := 16#7D24;
   // UNICODE_TO_GBK[25571] := 16#BC91;
   // UNICODE_TO_GBK[25572] := 16#7D25;
   // UNICODE_TO_GBK[25573] := 16#BC92;
   // UNICODE_TO_GBK[25574] := 16#7D26;
   // UNICODE_TO_GBK[25575] := 16#BC93;
   // UNICODE_TO_GBK[25576] := 16#7D27;
   // UNICODE_TO_GBK[25577] := 16#BDF4;
   // UNICODE_TO_GBK[25578] := 16#7D28;
   // UNICODE_TO_GBK[25579] := 16#BC94;
   // UNICODE_TO_GBK[25580] := 16#7D29;
   // UNICODE_TO_GBK[25581] := 16#BC95;
   // UNICODE_TO_GBK[25582] := 16#7D2A;
   // UNICODE_TO_GBK[25583] := 16#BC96;
   // UNICODE_TO_GBK[25584] := 16#7D2B;
   // UNICODE_TO_GBK[25585] := 16#D7CF;
   // UNICODE_TO_GBK[25586] := 16#7D2C;
   // UNICODE_TO_GBK[25587] := 16#BC97;
   // UNICODE_TO_GBK[25588] := 16#7D2D;
   // UNICODE_TO_GBK[25589] := 16#BC98;
   // UNICODE_TO_GBK[25590] := 16#7D2E;
   // UNICODE_TO_GBK[25591] := 16#BC99;
   // UNICODE_TO_GBK[25592] := 16#7D2F;
   // UNICODE_TO_GBK[25593] := 16#C0DB;
   // UNICODE_TO_GBK[25594] := 16#7D30;
   // UNICODE_TO_GBK[25595] := 16#BC9A;
   // UNICODE_TO_GBK[25596] := 16#7D31;
   // UNICODE_TO_GBK[25597] := 16#BC9B;
   // UNICODE_TO_GBK[25598] := 16#7D32;
   // UNICODE_TO_GBK[25599] := 16#BC9C;
   // UNICODE_TO_GBK[25600] := 16#7D33;
   // UNICODE_TO_GBK[25601] := 16#BC9D;
   // UNICODE_TO_GBK[25602] := 16#7D34;
   // UNICODE_TO_GBK[25603] := 16#BC9E;
   // UNICODE_TO_GBK[25604] := 16#7D35;
   // UNICODE_TO_GBK[25605] := 16#BC9F;
   // UNICODE_TO_GBK[25606] := 16#7D36;
   // UNICODE_TO_GBK[25607] := 16#BCA0;
   // UNICODE_TO_GBK[25608] := 16#7D37;
   // UNICODE_TO_GBK[25609] := 16#BD40;
   // UNICODE_TO_GBK[25610] := 16#7D38;
   // UNICODE_TO_GBK[25611] := 16#BD41;
   // UNICODE_TO_GBK[25612] := 16#7D39;
   // UNICODE_TO_GBK[25613] := 16#BD42;
   // UNICODE_TO_GBK[25614] := 16#7D3A;
   // UNICODE_TO_GBK[25615] := 16#BD43;
   // UNICODE_TO_GBK[25616] := 16#7D3B;
   // UNICODE_TO_GBK[25617] := 16#BD44;
   // UNICODE_TO_GBK[25618] := 16#7D3C;
   // UNICODE_TO_GBK[25619] := 16#BD45;
   // UNICODE_TO_GBK[25620] := 16#7D3D;
   // UNICODE_TO_GBK[25621] := 16#BD46;
   // UNICODE_TO_GBK[25622] := 16#7D3E;
   // UNICODE_TO_GBK[25623] := 16#BD47;
   // UNICODE_TO_GBK[25624] := 16#7D3F;
   // UNICODE_TO_GBK[25625] := 16#BD48;
   // UNICODE_TO_GBK[25626] := 16#7D40;
   // UNICODE_TO_GBK[25627] := 16#BD49;
   // UNICODE_TO_GBK[25628] := 16#7D41;
   // UNICODE_TO_GBK[25629] := 16#BD4A;
   // UNICODE_TO_GBK[25630] := 16#7D42;
   // UNICODE_TO_GBK[25631] := 16#BD4B;
   // UNICODE_TO_GBK[25632] := 16#7D43;
   // UNICODE_TO_GBK[25633] := 16#BD4C;
   // UNICODE_TO_GBK[25634] := 16#7D44;
   // UNICODE_TO_GBK[25635] := 16#BD4D;
   // UNICODE_TO_GBK[25636] := 16#7D45;
   // UNICODE_TO_GBK[25637] := 16#BD4E;
   // UNICODE_TO_GBK[25638] := 16#7D46;
   // UNICODE_TO_GBK[25639] := 16#BD4F;
   // UNICODE_TO_GBK[25640] := 16#7D47;
   // UNICODE_TO_GBK[25641] := 16#BD50;
   // UNICODE_TO_GBK[25642] := 16#7D48;
   // UNICODE_TO_GBK[25643] := 16#BD51;
   // UNICODE_TO_GBK[25644] := 16#7D49;
   // UNICODE_TO_GBK[25645] := 16#BD52;
   // UNICODE_TO_GBK[25646] := 16#7D4A;
   // UNICODE_TO_GBK[25647] := 16#BD53;
   // UNICODE_TO_GBK[25648] := 16#7D4B;
   // UNICODE_TO_GBK[25649] := 16#BD54;
   // UNICODE_TO_GBK[25650] := 16#7D4C;
   // UNICODE_TO_GBK[25651] := 16#BD55;
   // UNICODE_TO_GBK[25652] := 16#7D4D;
   // UNICODE_TO_GBK[25653] := 16#BD56;
   // UNICODE_TO_GBK[25654] := 16#7D4E;
   // UNICODE_TO_GBK[25655] := 16#BD57;
   // UNICODE_TO_GBK[25656] := 16#7D4F;
   // UNICODE_TO_GBK[25657] := 16#BD58;
   // UNICODE_TO_GBK[25658] := 16#7D50;
   // UNICODE_TO_GBK[25659] := 16#BD59;
   // UNICODE_TO_GBK[25660] := 16#7D51;
   // UNICODE_TO_GBK[25661] := 16#BD5A;
   // UNICODE_TO_GBK[25662] := 16#7D52;
   // UNICODE_TO_GBK[25663] := 16#BD5B;
   // UNICODE_TO_GBK[25664] := 16#7D53;
   // UNICODE_TO_GBK[25665] := 16#BD5C;
   // UNICODE_TO_GBK[25666] := 16#7D54;
   // UNICODE_TO_GBK[25667] := 16#BD5D;
   // UNICODE_TO_GBK[25668] := 16#7D55;
   // UNICODE_TO_GBK[25669] := 16#BD5E;
   // UNICODE_TO_GBK[25670] := 16#7D56;
   // UNICODE_TO_GBK[25671] := 16#BD5F;
   // UNICODE_TO_GBK[25672] := 16#7D57;
   // UNICODE_TO_GBK[25673] := 16#BD60;
   // UNICODE_TO_GBK[25674] := 16#7D58;
   // UNICODE_TO_GBK[25675] := 16#BD61;
   // UNICODE_TO_GBK[25676] := 16#7D59;
   // UNICODE_TO_GBK[25677] := 16#BD62;
   // UNICODE_TO_GBK[25678] := 16#7D5A;
   // UNICODE_TO_GBK[25679] := 16#BD63;
   // UNICODE_TO_GBK[25680] := 16#7D5B;
   // UNICODE_TO_GBK[25681] := 16#BD64;
   // UNICODE_TO_GBK[25682] := 16#7D5C;
   // UNICODE_TO_GBK[25683] := 16#BD65;
   // UNICODE_TO_GBK[25684] := 16#7D5D;
   // UNICODE_TO_GBK[25685] := 16#BD66;
   // UNICODE_TO_GBK[25686] := 16#7D5E;
   // UNICODE_TO_GBK[25687] := 16#BD67;
   // UNICODE_TO_GBK[25688] := 16#7D5F;
   // UNICODE_TO_GBK[25689] := 16#BD68;
   // UNICODE_TO_GBK[25690] := 16#7D60;
   // UNICODE_TO_GBK[25691] := 16#BD69;
   // UNICODE_TO_GBK[25692] := 16#7D61;
   // UNICODE_TO_GBK[25693] := 16#BD6A;
   // UNICODE_TO_GBK[25694] := 16#7D62;
   // UNICODE_TO_GBK[25695] := 16#BD6B;
   // UNICODE_TO_GBK[25696] := 16#7D63;
   // UNICODE_TO_GBK[25697] := 16#BD6C;
   // UNICODE_TO_GBK[25698] := 16#7D64;
   // UNICODE_TO_GBK[25699] := 16#BD6D;
   // UNICODE_TO_GBK[25700] := 16#7D65;
   // UNICODE_TO_GBK[25701] := 16#BD6E;
   // UNICODE_TO_GBK[25702] := 16#7D66;
   // UNICODE_TO_GBK[25703] := 16#BD6F;
   // UNICODE_TO_GBK[25704] := 16#7D67;
   // UNICODE_TO_GBK[25705] := 16#BD70;
   // UNICODE_TO_GBK[25706] := 16#7D68;
   // UNICODE_TO_GBK[25707] := 16#BD71;
   // UNICODE_TO_GBK[25708] := 16#7D69;
   // UNICODE_TO_GBK[25709] := 16#BD72;
   // UNICODE_TO_GBK[25710] := 16#7D6A;
   // UNICODE_TO_GBK[25711] := 16#BD73;
   // UNICODE_TO_GBK[25712] := 16#7D6B;
   // UNICODE_TO_GBK[25713] := 16#BD74;
   // UNICODE_TO_GBK[25714] := 16#7D6C;
   // UNICODE_TO_GBK[25715] := 16#BD75;
   // UNICODE_TO_GBK[25716] := 16#7D6D;
   // UNICODE_TO_GBK[25717] := 16#BD76;
   // UNICODE_TO_GBK[25718] := 16#7D6E;
   // UNICODE_TO_GBK[25719] := 16#D0F5;
   // UNICODE_TO_GBK[25720] := 16#7D6F;
   // UNICODE_TO_GBK[25721] := 16#BD77;
   // UNICODE_TO_GBK[25722] := 16#7D70;
   // UNICODE_TO_GBK[25723] := 16#BD78;
   // UNICODE_TO_GBK[25724] := 16#7D71;
   // UNICODE_TO_GBK[25725] := 16#BD79;
   // UNICODE_TO_GBK[25726] := 16#7D72;
   // UNICODE_TO_GBK[25727] := 16#BD7A;
   // UNICODE_TO_GBK[25728] := 16#7D73;
   // UNICODE_TO_GBK[25729] := 16#BD7B;
   // UNICODE_TO_GBK[25730] := 16#7D74;
   // UNICODE_TO_GBK[25731] := 16#BD7C;
   // UNICODE_TO_GBK[25732] := 16#7D75;
   // UNICODE_TO_GBK[25733] := 16#BD7D;
   // UNICODE_TO_GBK[25734] := 16#7D76;
   // UNICODE_TO_GBK[25735] := 16#BD7E;
   // UNICODE_TO_GBK[25736] := 16#7D77;
   // UNICODE_TO_GBK[25737] := 16#F4EA;
   // UNICODE_TO_GBK[25738] := 16#7D78;
   // UNICODE_TO_GBK[25739] := 16#BD80;
   // UNICODE_TO_GBK[25740] := 16#7D79;
   // UNICODE_TO_GBK[25741] := 16#BD81;
   // UNICODE_TO_GBK[25742] := 16#7D7A;
   // UNICODE_TO_GBK[25743] := 16#BD82;
   // UNICODE_TO_GBK[25744] := 16#7D7B;
   // UNICODE_TO_GBK[25745] := 16#BD83;
   // UNICODE_TO_GBK[25746] := 16#7D7C;
   // UNICODE_TO_GBK[25747] := 16#BD84;
   // UNICODE_TO_GBK[25748] := 16#7D7D;
   // UNICODE_TO_GBK[25749] := 16#BD85;
   // UNICODE_TO_GBK[25750] := 16#7D7E;
   // UNICODE_TO_GBK[25751] := 16#BD86;
   // UNICODE_TO_GBK[25752] := 16#7D7F;
   // UNICODE_TO_GBK[25753] := 16#BD87;
   // UNICODE_TO_GBK[25754] := 16#7D80;
   // UNICODE_TO_GBK[25755] := 16#BD88;
   // UNICODE_TO_GBK[25756] := 16#7D81;
   // UNICODE_TO_GBK[25757] := 16#BD89;
   // UNICODE_TO_GBK[25758] := 16#7D82;
   // UNICODE_TO_GBK[25759] := 16#BD8A;
   // UNICODE_TO_GBK[25760] := 16#7D83;
   // UNICODE_TO_GBK[25761] := 16#BD8B;
   // UNICODE_TO_GBK[25762] := 16#7D84;
   // UNICODE_TO_GBK[25763] := 16#BD8C;
   // UNICODE_TO_GBK[25764] := 16#7D85;
   // UNICODE_TO_GBK[25765] := 16#BD8D;
   // UNICODE_TO_GBK[25766] := 16#7D86;
   // UNICODE_TO_GBK[25767] := 16#BD8E;
   // UNICODE_TO_GBK[25768] := 16#7D87;
   // UNICODE_TO_GBK[25769] := 16#BD8F;
   // UNICODE_TO_GBK[25770] := 16#7D88;
   // UNICODE_TO_GBK[25771] := 16#BD90;
   // UNICODE_TO_GBK[25772] := 16#7D89;
   // UNICODE_TO_GBK[25773] := 16#BD91;
   // UNICODE_TO_GBK[25774] := 16#7D8A;
   // UNICODE_TO_GBK[25775] := 16#BD92;
   // UNICODE_TO_GBK[25776] := 16#7D8B;
   // UNICODE_TO_GBK[25777] := 16#BD93;
   // UNICODE_TO_GBK[25778] := 16#7D8C;
   // UNICODE_TO_GBK[25779] := 16#BD94;
   // UNICODE_TO_GBK[25780] := 16#7D8D;
   // UNICODE_TO_GBK[25781] := 16#BD95;
   // UNICODE_TO_GBK[25782] := 16#7D8E;
   // UNICODE_TO_GBK[25783] := 16#BD96;
   // UNICODE_TO_GBK[25784] := 16#7D8F;
   // UNICODE_TO_GBK[25785] := 16#BD97;
   // UNICODE_TO_GBK[25786] := 16#7D90;
   // UNICODE_TO_GBK[25787] := 16#BD98;
   // UNICODE_TO_GBK[25788] := 16#7D91;
   // UNICODE_TO_GBK[25789] := 16#BD99;
   // UNICODE_TO_GBK[25790] := 16#7D92;
   // UNICODE_TO_GBK[25791] := 16#BD9A;
   // UNICODE_TO_GBK[25792] := 16#7D93;
   // UNICODE_TO_GBK[25793] := 16#BD9B;
   // UNICODE_TO_GBK[25794] := 16#7D94;
   // UNICODE_TO_GBK[25795] := 16#BD9C;
   // UNICODE_TO_GBK[25796] := 16#7D95;
   // UNICODE_TO_GBK[25797] := 16#BD9D;
   // UNICODE_TO_GBK[25798] := 16#7D96;
   // UNICODE_TO_GBK[25799] := 16#BD9E;
   // UNICODE_TO_GBK[25800] := 16#7D97;
   // UNICODE_TO_GBK[25801] := 16#BD9F;
   // UNICODE_TO_GBK[25802] := 16#7D98;
   // UNICODE_TO_GBK[25803] := 16#BDA0;
   // UNICODE_TO_GBK[25804] := 16#7D99;
   // UNICODE_TO_GBK[25805] := 16#BE40;
   // UNICODE_TO_GBK[25806] := 16#7D9A;
   // UNICODE_TO_GBK[25807] := 16#BE41;
   // UNICODE_TO_GBK[25808] := 16#7D9B;
   // UNICODE_TO_GBK[25809] := 16#BE42;
   // UNICODE_TO_GBK[25810] := 16#7D9C;
   // UNICODE_TO_GBK[25811] := 16#BE43;
   // UNICODE_TO_GBK[25812] := 16#7D9D;
   // UNICODE_TO_GBK[25813] := 16#BE44;
   // UNICODE_TO_GBK[25814] := 16#7D9E;
   // UNICODE_TO_GBK[25815] := 16#BE45;
   // UNICODE_TO_GBK[25816] := 16#7D9F;
   // UNICODE_TO_GBK[25817] := 16#BE46;
   // UNICODE_TO_GBK[25818] := 16#7DA0;
   // UNICODE_TO_GBK[25819] := 16#BE47;
   // UNICODE_TO_GBK[25820] := 16#7DA1;
   // UNICODE_TO_GBK[25821] := 16#BE48;
   // UNICODE_TO_GBK[25822] := 16#7DA2;
   // UNICODE_TO_GBK[25823] := 16#BE49;
   // UNICODE_TO_GBK[25824] := 16#7DA3;
   // UNICODE_TO_GBK[25825] := 16#BE4A;
   // UNICODE_TO_GBK[25826] := 16#7DA4;
   // UNICODE_TO_GBK[25827] := 16#BE4B;
   // UNICODE_TO_GBK[25828] := 16#7DA5;
   // UNICODE_TO_GBK[25829] := 16#BE4C;
   // UNICODE_TO_GBK[25830] := 16#7DA6;
   // UNICODE_TO_GBK[25831] := 16#F4EB;
   // UNICODE_TO_GBK[25832] := 16#7DA7;
   // UNICODE_TO_GBK[25833] := 16#BE4D;
   // UNICODE_TO_GBK[25834] := 16#7DA8;
   // UNICODE_TO_GBK[25835] := 16#BE4E;
   // UNICODE_TO_GBK[25836] := 16#7DA9;
   // UNICODE_TO_GBK[25837] := 16#BE4F;
   // UNICODE_TO_GBK[25838] := 16#7DAA;
   // UNICODE_TO_GBK[25839] := 16#BE50;
   // UNICODE_TO_GBK[25840] := 16#7DAB;
   // UNICODE_TO_GBK[25841] := 16#BE51;
   // UNICODE_TO_GBK[25842] := 16#7DAC;
   // UNICODE_TO_GBK[25843] := 16#BE52;
   // UNICODE_TO_GBK[25844] := 16#7DAD;
   // UNICODE_TO_GBK[25845] := 16#BE53;
   // UNICODE_TO_GBK[25846] := 16#7DAE;
   // UNICODE_TO_GBK[25847] := 16#F4EC;
   // UNICODE_TO_GBK[25848] := 16#7DAF;
   // UNICODE_TO_GBK[25849] := 16#BE54;
   // UNICODE_TO_GBK[25850] := 16#7DB0;
   // UNICODE_TO_GBK[25851] := 16#BE55;
   // UNICODE_TO_GBK[25852] := 16#7DB1;
   // UNICODE_TO_GBK[25853] := 16#BE56;
   // UNICODE_TO_GBK[25854] := 16#7DB2;
   // UNICODE_TO_GBK[25855] := 16#BE57;
   // UNICODE_TO_GBK[25856] := 16#7DB3;
   // UNICODE_TO_GBK[25857] := 16#BE58;
   // UNICODE_TO_GBK[25858] := 16#7DB4;
   // UNICODE_TO_GBK[25859] := 16#BE59;
   // UNICODE_TO_GBK[25860] := 16#7DB5;
   // UNICODE_TO_GBK[25861] := 16#BE5A;
   // UNICODE_TO_GBK[25862] := 16#7DB6;
   // UNICODE_TO_GBK[25863] := 16#BE5B;
   // UNICODE_TO_GBK[25864] := 16#7DB7;
   // UNICODE_TO_GBK[25865] := 16#BE5C;
   // UNICODE_TO_GBK[25866] := 16#7DB8;
   // UNICODE_TO_GBK[25867] := 16#BE5D;
   // UNICODE_TO_GBK[25868] := 16#7DB9;
   // UNICODE_TO_GBK[25869] := 16#BE5E;
   // UNICODE_TO_GBK[25870] := 16#7DBA;
   // UNICODE_TO_GBK[25871] := 16#BE5F;
   // UNICODE_TO_GBK[25872] := 16#7DBB;
   // UNICODE_TO_GBK[25873] := 16#BE60;
   // UNICODE_TO_GBK[25874] := 16#7DBC;
   // UNICODE_TO_GBK[25875] := 16#BE61;
   // UNICODE_TO_GBK[25876] := 16#7DBD;
   // UNICODE_TO_GBK[25877] := 16#BE62;
   // UNICODE_TO_GBK[25878] := 16#7DBE;
   // UNICODE_TO_GBK[25879] := 16#BE63;
   // UNICODE_TO_GBK[25880] := 16#7DBF;
   // UNICODE_TO_GBK[25881] := 16#BE64;
   // UNICODE_TO_GBK[25882] := 16#7DC0;
   // UNICODE_TO_GBK[25883] := 16#BE65;
   // UNICODE_TO_GBK[25884] := 16#7DC1;
   // UNICODE_TO_GBK[25885] := 16#BE66;
   // UNICODE_TO_GBK[25886] := 16#7DC2;
   // UNICODE_TO_GBK[25887] := 16#BE67;
   // UNICODE_TO_GBK[25888] := 16#7DC3;
   // UNICODE_TO_GBK[25889] := 16#BE68;
   // UNICODE_TO_GBK[25890] := 16#7DC4;
   // UNICODE_TO_GBK[25891] := 16#BE69;
   // UNICODE_TO_GBK[25892] := 16#7DC5;
   // UNICODE_TO_GBK[25893] := 16#BE6A;
   // UNICODE_TO_GBK[25894] := 16#7DC6;
   // UNICODE_TO_GBK[25895] := 16#BE6B;
   // UNICODE_TO_GBK[25896] := 16#7DC7;
   // UNICODE_TO_GBK[25897] := 16#BE6C;
   // UNICODE_TO_GBK[25898] := 16#7DC8;
   // UNICODE_TO_GBK[25899] := 16#BE6D;
   // UNICODE_TO_GBK[25900] := 16#7DC9;
   // UNICODE_TO_GBK[25901] := 16#BE6E;
   // UNICODE_TO_GBK[25902] := 16#7DCA;
   // UNICODE_TO_GBK[25903] := 16#BE6F;
   // UNICODE_TO_GBK[25904] := 16#7DCB;
   // UNICODE_TO_GBK[25905] := 16#BE70;
   // UNICODE_TO_GBK[25906] := 16#7DCC;
   // UNICODE_TO_GBK[25907] := 16#BE71;
   // UNICODE_TO_GBK[25908] := 16#7DCD;
   // UNICODE_TO_GBK[25909] := 16#BE72;
   // UNICODE_TO_GBK[25910] := 16#7DCE;
   // UNICODE_TO_GBK[25911] := 16#BE73;
   // UNICODE_TO_GBK[25912] := 16#7DCF;
   // UNICODE_TO_GBK[25913] := 16#BE74;
   // UNICODE_TO_GBK[25914] := 16#7DD0;
   // UNICODE_TO_GBK[25915] := 16#BE75;
   // UNICODE_TO_GBK[25916] := 16#7DD1;
   // UNICODE_TO_GBK[25917] := 16#BE76;
   // UNICODE_TO_GBK[25918] := 16#7DD2;
   // UNICODE_TO_GBK[25919] := 16#BE77;
   // UNICODE_TO_GBK[25920] := 16#7DD3;
   // UNICODE_TO_GBK[25921] := 16#BE78;
   // UNICODE_TO_GBK[25922] := 16#7DD4;
   // UNICODE_TO_GBK[25923] := 16#BE79;
   // UNICODE_TO_GBK[25924] := 16#7DD5;
   // UNICODE_TO_GBK[25925] := 16#BE7A;
   // UNICODE_TO_GBK[25926] := 16#7DD6;
   // UNICODE_TO_GBK[25927] := 16#BE7B;
   // UNICODE_TO_GBK[25928] := 16#7DD7;
   // UNICODE_TO_GBK[25929] := 16#BE7C;
   // UNICODE_TO_GBK[25930] := 16#7DD8;
   // UNICODE_TO_GBK[25931] := 16#BE7D;
   // UNICODE_TO_GBK[25932] := 16#7DD9;
   // UNICODE_TO_GBK[25933] := 16#BE7E;
   // UNICODE_TO_GBK[25934] := 16#7DDA;
   // UNICODE_TO_GBK[25935] := 16#BE80;
   // UNICODE_TO_GBK[25936] := 16#7DDB;
   // UNICODE_TO_GBK[25937] := 16#BE81;
   // UNICODE_TO_GBK[25938] := 16#7DDC;
   // UNICODE_TO_GBK[25939] := 16#BE82;
   // UNICODE_TO_GBK[25940] := 16#7DDD;
   // UNICODE_TO_GBK[25941] := 16#BE83;
   // UNICODE_TO_GBK[25942] := 16#7DDE;
   // UNICODE_TO_GBK[25943] := 16#BE84;
   // UNICODE_TO_GBK[25944] := 16#7DDF;
   // UNICODE_TO_GBK[25945] := 16#BE85;
   // UNICODE_TO_GBK[25946] := 16#7DE0;
   // UNICODE_TO_GBK[25947] := 16#BE86;
   // UNICODE_TO_GBK[25948] := 16#7DE1;
   // UNICODE_TO_GBK[25949] := 16#BE87;
   // UNICODE_TO_GBK[25950] := 16#7DE2;
   // UNICODE_TO_GBK[25951] := 16#BE88;
   // UNICODE_TO_GBK[25952] := 16#7DE3;
   // UNICODE_TO_GBK[25953] := 16#BE89;
   // UNICODE_TO_GBK[25954] := 16#7DE4;
   // UNICODE_TO_GBK[25955] := 16#BE8A;
   // UNICODE_TO_GBK[25956] := 16#7DE5;
   // UNICODE_TO_GBK[25957] := 16#BE8B;
   // UNICODE_TO_GBK[25958] := 16#7DE6;
   // UNICODE_TO_GBK[25959] := 16#BE8C;
   // UNICODE_TO_GBK[25960] := 16#7DE7;
   // UNICODE_TO_GBK[25961] := 16#BE8D;
   // UNICODE_TO_GBK[25962] := 16#7DE8;
   // UNICODE_TO_GBK[25963] := 16#BE8E;
   // UNICODE_TO_GBK[25964] := 16#7DE9;
   // UNICODE_TO_GBK[25965] := 16#BE8F;
   // UNICODE_TO_GBK[25966] := 16#7DEA;
   // UNICODE_TO_GBK[25967] := 16#BE90;
   // UNICODE_TO_GBK[25968] := 16#7DEB;
   // UNICODE_TO_GBK[25969] := 16#BE91;
   // UNICODE_TO_GBK[25970] := 16#7DEC;
   // UNICODE_TO_GBK[25971] := 16#BE92;
   // UNICODE_TO_GBK[25972] := 16#7DED;
   // UNICODE_TO_GBK[25973] := 16#BE93;
   // UNICODE_TO_GBK[25974] := 16#7DEE;
   // UNICODE_TO_GBK[25975] := 16#BE94;
   // UNICODE_TO_GBK[25976] := 16#7DEF;
   // UNICODE_TO_GBK[25977] := 16#BE95;
   // UNICODE_TO_GBK[25978] := 16#7DF0;
   // UNICODE_TO_GBK[25979] := 16#BE96;
   // UNICODE_TO_GBK[25980] := 16#7DF1;
   // UNICODE_TO_GBK[25981] := 16#BE97;
   // UNICODE_TO_GBK[25982] := 16#7DF2;
   // UNICODE_TO_GBK[25983] := 16#BE98;
   // UNICODE_TO_GBK[25984] := 16#7DF3;
   // UNICODE_TO_GBK[25985] := 16#BE99;
   // UNICODE_TO_GBK[25986] := 16#7DF4;
   // UNICODE_TO_GBK[25987] := 16#BE9A;
   // UNICODE_TO_GBK[25988] := 16#7DF5;
   // UNICODE_TO_GBK[25989] := 16#BE9B;
   // UNICODE_TO_GBK[25990] := 16#7DF6;
   // UNICODE_TO_GBK[25991] := 16#BE9C;
   // UNICODE_TO_GBK[25992] := 16#7DF7;
   // UNICODE_TO_GBK[25993] := 16#BE9D;
   // UNICODE_TO_GBK[25994] := 16#7DF8;
   // UNICODE_TO_GBK[25995] := 16#BE9E;
   // UNICODE_TO_GBK[25996] := 16#7DF9;
   // UNICODE_TO_GBK[25997] := 16#BE9F;
   // UNICODE_TO_GBK[25998] := 16#7DFA;
   // UNICODE_TO_GBK[25999] := 16#BEA0;
   // UNICODE_TO_GBK[26000] := 16#7DFB;
   // UNICODE_TO_GBK[26001] := 16#BF40;
   // UNICODE_TO_GBK[26002] := 16#7DFC;
   // UNICODE_TO_GBK[26003] := 16#BF41;
   // UNICODE_TO_GBK[26004] := 16#7DFD;
   // UNICODE_TO_GBK[26005] := 16#BF42;
   // UNICODE_TO_GBK[26006] := 16#7DFE;
   // UNICODE_TO_GBK[26007] := 16#BF43;
   // UNICODE_TO_GBK[26008] := 16#7DFF;
   // UNICODE_TO_GBK[26009] := 16#BF44;
   // UNICODE_TO_GBK[26010] := 16#7E00;
   // UNICODE_TO_GBK[26011] := 16#BF45;
   // UNICODE_TO_GBK[26012] := 16#7E01;
   // UNICODE_TO_GBK[26013] := 16#BF46;
   // UNICODE_TO_GBK[26014] := 16#7E02;
   // UNICODE_TO_GBK[26015] := 16#BF47;
   // UNICODE_TO_GBK[26016] := 16#7E03;
   // UNICODE_TO_GBK[26017] := 16#BF48;
   // UNICODE_TO_GBK[26018] := 16#7E04;
   // UNICODE_TO_GBK[26019] := 16#BF49;
   // UNICODE_TO_GBK[26020] := 16#7E05;
   // UNICODE_TO_GBK[26021] := 16#BF4A;
   // UNICODE_TO_GBK[26022] := 16#7E06;
   // UNICODE_TO_GBK[26023] := 16#BF4B;
   // UNICODE_TO_GBK[26024] := 16#7E07;
   // UNICODE_TO_GBK[26025] := 16#BF4C;
   // UNICODE_TO_GBK[26026] := 16#7E08;
   // UNICODE_TO_GBK[26027] := 16#BF4D;
   // UNICODE_TO_GBK[26028] := 16#7E09;
   // UNICODE_TO_GBK[26029] := 16#BF4E;
   // UNICODE_TO_GBK[26030] := 16#7E0A;
   // UNICODE_TO_GBK[26031] := 16#BF4F;
   // UNICODE_TO_GBK[26032] := 16#7E0B;
   // UNICODE_TO_GBK[26033] := 16#BF50;
   // UNICODE_TO_GBK[26034] := 16#7E0C;
   // UNICODE_TO_GBK[26035] := 16#BF51;
   // UNICODE_TO_GBK[26036] := 16#7E0D;
   // UNICODE_TO_GBK[26037] := 16#BF52;
   // UNICODE_TO_GBK[26038] := 16#7E0E;
   // UNICODE_TO_GBK[26039] := 16#BF53;
   // UNICODE_TO_GBK[26040] := 16#7E0F;
   // UNICODE_TO_GBK[26041] := 16#BF54;
   // UNICODE_TO_GBK[26042] := 16#7E10;
   // UNICODE_TO_GBK[26043] := 16#BF55;
   // UNICODE_TO_GBK[26044] := 16#7E11;
   // UNICODE_TO_GBK[26045] := 16#BF56;
   // UNICODE_TO_GBK[26046] := 16#7E12;
   // UNICODE_TO_GBK[26047] := 16#BF57;
   // UNICODE_TO_GBK[26048] := 16#7E13;
   // UNICODE_TO_GBK[26049] := 16#BF58;
   // UNICODE_TO_GBK[26050] := 16#7E14;
   // UNICODE_TO_GBK[26051] := 16#BF59;
   // UNICODE_TO_GBK[26052] := 16#7E15;
   // UNICODE_TO_GBK[26053] := 16#BF5A;
   // UNICODE_TO_GBK[26054] := 16#7E16;
   // UNICODE_TO_GBK[26055] := 16#BF5B;
   // UNICODE_TO_GBK[26056] := 16#7E17;
   // UNICODE_TO_GBK[26057] := 16#BF5C;
   // UNICODE_TO_GBK[26058] := 16#7E18;
   // UNICODE_TO_GBK[26059] := 16#BF5D;
   // UNICODE_TO_GBK[26060] := 16#7E19;
   // UNICODE_TO_GBK[26061] := 16#BF5E;
   // UNICODE_TO_GBK[26062] := 16#7E1A;
   // UNICODE_TO_GBK[26063] := 16#BF5F;
   // UNICODE_TO_GBK[26064] := 16#7E1B;
   // UNICODE_TO_GBK[26065] := 16#BF60;
   // UNICODE_TO_GBK[26066] := 16#7E1C;
   // UNICODE_TO_GBK[26067] := 16#BF61;
   // UNICODE_TO_GBK[26068] := 16#7E1D;
   // UNICODE_TO_GBK[26069] := 16#BF62;
   // UNICODE_TO_GBK[26070] := 16#7E1E;
   // UNICODE_TO_GBK[26071] := 16#BF63;
   // UNICODE_TO_GBK[26072] := 16#7E1F;
   // UNICODE_TO_GBK[26073] := 16#BF64;
   // UNICODE_TO_GBK[26074] := 16#7E20;
   // UNICODE_TO_GBK[26075] := 16#BF65;
   // UNICODE_TO_GBK[26076] := 16#7E21;
   // UNICODE_TO_GBK[26077] := 16#BF66;
   // UNICODE_TO_GBK[26078] := 16#7E22;
   // UNICODE_TO_GBK[26079] := 16#BF67;
   // UNICODE_TO_GBK[26080] := 16#7E23;
   // UNICODE_TO_GBK[26081] := 16#BF68;
   // UNICODE_TO_GBK[26082] := 16#7E24;
   // UNICODE_TO_GBK[26083] := 16#BF69;
   // UNICODE_TO_GBK[26084] := 16#7E25;
   // UNICODE_TO_GBK[26085] := 16#BF6A;
   // UNICODE_TO_GBK[26086] := 16#7E26;
   // UNICODE_TO_GBK[26087] := 16#BF6B;
   // UNICODE_TO_GBK[26088] := 16#7E27;
   // UNICODE_TO_GBK[26089] := 16#BF6C;
   // UNICODE_TO_GBK[26090] := 16#7E28;
   // UNICODE_TO_GBK[26091] := 16#BF6D;
   // UNICODE_TO_GBK[26092] := 16#7E29;
   // UNICODE_TO_GBK[26093] := 16#BF6E;
   // UNICODE_TO_GBK[26094] := 16#7E2A;
   // UNICODE_TO_GBK[26095] := 16#BF6F;
   // UNICODE_TO_GBK[26096] := 16#7E2B;
   // UNICODE_TO_GBK[26097] := 16#BF70;
   // UNICODE_TO_GBK[26098] := 16#7E2C;
   // UNICODE_TO_GBK[26099] := 16#BF71;
   // UNICODE_TO_GBK[26100] := 16#7E2D;
   // UNICODE_TO_GBK[26101] := 16#BF72;
   // UNICODE_TO_GBK[26102] := 16#7E2E;
   // UNICODE_TO_GBK[26103] := 16#BF73;
   // UNICODE_TO_GBK[26104] := 16#7E2F;
   // UNICODE_TO_GBK[26105] := 16#BF74;
   // UNICODE_TO_GBK[26106] := 16#7E30;
   // UNICODE_TO_GBK[26107] := 16#BF75;
   // UNICODE_TO_GBK[26108] := 16#7E31;
   // UNICODE_TO_GBK[26109] := 16#BF76;
   // UNICODE_TO_GBK[26110] := 16#7E32;
   // UNICODE_TO_GBK[26111] := 16#BF77;
   // UNICODE_TO_GBK[26112] := 16#7E33;
   // UNICODE_TO_GBK[26113] := 16#BF78;
   // UNICODE_TO_GBK[26114] := 16#7E34;
   // UNICODE_TO_GBK[26115] := 16#BF79;
   // UNICODE_TO_GBK[26116] := 16#7E35;
   // UNICODE_TO_GBK[26117] := 16#BF7A;
   // UNICODE_TO_GBK[26118] := 16#7E36;
   // UNICODE_TO_GBK[26119] := 16#BF7B;
   // UNICODE_TO_GBK[26120] := 16#7E37;
   // UNICODE_TO_GBK[26121] := 16#BF7C;
   // UNICODE_TO_GBK[26122] := 16#7E38;
   // UNICODE_TO_GBK[26123] := 16#BF7D;
   // UNICODE_TO_GBK[26124] := 16#7E39;
   // UNICODE_TO_GBK[26125] := 16#BF7E;
   // UNICODE_TO_GBK[26126] := 16#7E3A;
   // UNICODE_TO_GBK[26127] := 16#BF80;
   // UNICODE_TO_GBK[26128] := 16#7E3B;
   // UNICODE_TO_GBK[26129] := 16#F7E3;
   // UNICODE_TO_GBK[26130] := 16#7E3C;
   // UNICODE_TO_GBK[26131] := 16#BF81;
   // UNICODE_TO_GBK[26132] := 16#7E3D;
   // UNICODE_TO_GBK[26133] := 16#BF82;
   // UNICODE_TO_GBK[26134] := 16#7E3E;
   // UNICODE_TO_GBK[26135] := 16#BF83;
   // UNICODE_TO_GBK[26136] := 16#7E3F;
   // UNICODE_TO_GBK[26137] := 16#BF84;
   // UNICODE_TO_GBK[26138] := 16#7E40;
   // UNICODE_TO_GBK[26139] := 16#BF85;
   // UNICODE_TO_GBK[26140] := 16#7E41;
   // UNICODE_TO_GBK[26141] := 16#B7B1;
   // UNICODE_TO_GBK[26142] := 16#7E42;
   // UNICODE_TO_GBK[26143] := 16#BF86;
   // UNICODE_TO_GBK[26144] := 16#7E43;
   // UNICODE_TO_GBK[26145] := 16#BF87;
   // UNICODE_TO_GBK[26146] := 16#7E44;
   // UNICODE_TO_GBK[26147] := 16#BF88;
   // UNICODE_TO_GBK[26148] := 16#7E45;
   // UNICODE_TO_GBK[26149] := 16#BF89;
   // UNICODE_TO_GBK[26150] := 16#7E46;
   // UNICODE_TO_GBK[26151] := 16#BF8A;
   // UNICODE_TO_GBK[26152] := 16#7E47;
   // UNICODE_TO_GBK[26153] := 16#F4ED;
   // UNICODE_TO_GBK[26154] := 16#7E48;
   // UNICODE_TO_GBK[26155] := 16#BF8B;
   // UNICODE_TO_GBK[26156] := 16#7E49;
   // UNICODE_TO_GBK[26157] := 16#BF8C;
   // UNICODE_TO_GBK[26158] := 16#7E4A;
   // UNICODE_TO_GBK[26159] := 16#BF8D;
   // UNICODE_TO_GBK[26160] := 16#7E4B;
   // UNICODE_TO_GBK[26161] := 16#BF8E;
   // UNICODE_TO_GBK[26162] := 16#7E4C;
   // UNICODE_TO_GBK[26163] := 16#BF8F;
   // UNICODE_TO_GBK[26164] := 16#7E4D;
   // UNICODE_TO_GBK[26165] := 16#BF90;
   // UNICODE_TO_GBK[26166] := 16#7E4E;
   // UNICODE_TO_GBK[26167] := 16#BF91;
   // UNICODE_TO_GBK[26168] := 16#7E4F;
   // UNICODE_TO_GBK[26169] := 16#BF92;
   // UNICODE_TO_GBK[26170] := 16#7E50;
   // UNICODE_TO_GBK[26171] := 16#BF93;
   // UNICODE_TO_GBK[26172] := 16#7E51;
   // UNICODE_TO_GBK[26173] := 16#BF94;
   // UNICODE_TO_GBK[26174] := 16#7E52;
   // UNICODE_TO_GBK[26175] := 16#BF95;
   // UNICODE_TO_GBK[26176] := 16#7E53;
   // UNICODE_TO_GBK[26177] := 16#BF96;
   // UNICODE_TO_GBK[26178] := 16#7E54;
   // UNICODE_TO_GBK[26179] := 16#BF97;
   // UNICODE_TO_GBK[26180] := 16#7E55;
   // UNICODE_TO_GBK[26181] := 16#BF98;
   // UNICODE_TO_GBK[26182] := 16#7E56;
   // UNICODE_TO_GBK[26183] := 16#BF99;
   // UNICODE_TO_GBK[26184] := 16#7E57;
   // UNICODE_TO_GBK[26185] := 16#BF9A;
   // UNICODE_TO_GBK[26186] := 16#7E58;
   // UNICODE_TO_GBK[26187] := 16#BF9B;
   // UNICODE_TO_GBK[26188] := 16#7E59;
   // UNICODE_TO_GBK[26189] := 16#BF9C;
   // UNICODE_TO_GBK[26190] := 16#7E5A;
   // UNICODE_TO_GBK[26191] := 16#BF9D;
   // UNICODE_TO_GBK[26192] := 16#7E5B;
   // UNICODE_TO_GBK[26193] := 16#BF9E;
   // UNICODE_TO_GBK[26194] := 16#7E5C;
   // UNICODE_TO_GBK[26195] := 16#BF9F;
   // UNICODE_TO_GBK[26196] := 16#7E5D;
   // UNICODE_TO_GBK[26197] := 16#BFA0;
   // UNICODE_TO_GBK[26198] := 16#7E5E;
   // UNICODE_TO_GBK[26199] := 16#C040;
   // UNICODE_TO_GBK[26200] := 16#7E5F;
   // UNICODE_TO_GBK[26201] := 16#C041;
   // UNICODE_TO_GBK[26202] := 16#7E60;
   // UNICODE_TO_GBK[26203] := 16#C042;
   // UNICODE_TO_GBK[26204] := 16#7E61;
   // UNICODE_TO_GBK[26205] := 16#C043;
   // UNICODE_TO_GBK[26206] := 16#7E62;
   // UNICODE_TO_GBK[26207] := 16#C044;
   // UNICODE_TO_GBK[26208] := 16#7E63;
   // UNICODE_TO_GBK[26209] := 16#C045;
   // UNICODE_TO_GBK[26210] := 16#7E64;
   // UNICODE_TO_GBK[26211] := 16#C046;
   // UNICODE_TO_GBK[26212] := 16#7E65;
   // UNICODE_TO_GBK[26213] := 16#C047;
   // UNICODE_TO_GBK[26214] := 16#7E66;
   // UNICODE_TO_GBK[26215] := 16#C048;
   // UNICODE_TO_GBK[26216] := 16#7E67;
   // UNICODE_TO_GBK[26217] := 16#C049;
   // UNICODE_TO_GBK[26218] := 16#7E68;
   // UNICODE_TO_GBK[26219] := 16#C04A;
   // UNICODE_TO_GBK[26220] := 16#7E69;
   // UNICODE_TO_GBK[26221] := 16#C04B;
   // UNICODE_TO_GBK[26222] := 16#7E6A;
   // UNICODE_TO_GBK[26223] := 16#C04C;
   // UNICODE_TO_GBK[26224] := 16#7E6B;
   // UNICODE_TO_GBK[26225] := 16#C04D;
   // UNICODE_TO_GBK[26226] := 16#7E6C;
   // UNICODE_TO_GBK[26227] := 16#C04E;
   // UNICODE_TO_GBK[26228] := 16#7E6D;
   // UNICODE_TO_GBK[26229] := 16#C04F;
   // UNICODE_TO_GBK[26230] := 16#7E6E;
   // UNICODE_TO_GBK[26231] := 16#C050;
   // UNICODE_TO_GBK[26232] := 16#7E6F;
   // UNICODE_TO_GBK[26233] := 16#C051;
   // UNICODE_TO_GBK[26234] := 16#7E70;
   // UNICODE_TO_GBK[26235] := 16#C052;
   // UNICODE_TO_GBK[26236] := 16#7E71;
   // UNICODE_TO_GBK[26237] := 16#C053;
   // UNICODE_TO_GBK[26238] := 16#7E72;
   // UNICODE_TO_GBK[26239] := 16#C054;
   // UNICODE_TO_GBK[26240] := 16#7E73;
   // UNICODE_TO_GBK[26241] := 16#C055;
   // UNICODE_TO_GBK[26242] := 16#7E74;
   // UNICODE_TO_GBK[26243] := 16#C056;
   // UNICODE_TO_GBK[26244] := 16#7E75;
   // UNICODE_TO_GBK[26245] := 16#C057;
   // UNICODE_TO_GBK[26246] := 16#7E76;
   // UNICODE_TO_GBK[26247] := 16#C058;
   // UNICODE_TO_GBK[26248] := 16#7E77;
   // UNICODE_TO_GBK[26249] := 16#C059;
   // UNICODE_TO_GBK[26250] := 16#7E78;
   // UNICODE_TO_GBK[26251] := 16#C05A;
   // UNICODE_TO_GBK[26252] := 16#7E79;
   // UNICODE_TO_GBK[26253] := 16#C05B;
   // UNICODE_TO_GBK[26254] := 16#7E7A;
   // UNICODE_TO_GBK[26255] := 16#C05C;
   // UNICODE_TO_GBK[26256] := 16#7E7B;
   // UNICODE_TO_GBK[26257] := 16#C05D;
   // UNICODE_TO_GBK[26258] := 16#7E7C;
   // UNICODE_TO_GBK[26259] := 16#C05E;
   // UNICODE_TO_GBK[26260] := 16#7E7D;
   // UNICODE_TO_GBK[26261] := 16#C05F;
   // UNICODE_TO_GBK[26262] := 16#7E7E;
   // UNICODE_TO_GBK[26263] := 16#C060;
   // UNICODE_TO_GBK[26264] := 16#7E7F;
   // UNICODE_TO_GBK[26265] := 16#C061;
   // UNICODE_TO_GBK[26266] := 16#7E80;
   // UNICODE_TO_GBK[26267] := 16#C062;
   // UNICODE_TO_GBK[26268] := 16#7E81;
   // UNICODE_TO_GBK[26269] := 16#C063;
   // UNICODE_TO_GBK[26270] := 16#7E82;
   // UNICODE_TO_GBK[26271] := 16#D7EB;
   // UNICODE_TO_GBK[26272] := 16#7E83;
   // UNICODE_TO_GBK[26273] := 16#C064;
   // UNICODE_TO_GBK[26274] := 16#7E84;
   // UNICODE_TO_GBK[26275] := 16#C065;
   // UNICODE_TO_GBK[26276] := 16#7E85;
   // UNICODE_TO_GBK[26277] := 16#C066;
   // UNICODE_TO_GBK[26278] := 16#7E86;
   // UNICODE_TO_GBK[26279] := 16#C067;
   // UNICODE_TO_GBK[26280] := 16#7E87;
   // UNICODE_TO_GBK[26281] := 16#C068;
   // UNICODE_TO_GBK[26282] := 16#7E88;
   // UNICODE_TO_GBK[26283] := 16#C069;
   // UNICODE_TO_GBK[26284] := 16#7E89;
   // UNICODE_TO_GBK[26285] := 16#C06A;
   // UNICODE_TO_GBK[26286] := 16#7E8A;
   // UNICODE_TO_GBK[26287] := 16#C06B;
   // UNICODE_TO_GBK[26288] := 16#7E8B;
   // UNICODE_TO_GBK[26289] := 16#C06C;
   // UNICODE_TO_GBK[26290] := 16#7E8C;
   // UNICODE_TO_GBK[26291] := 16#C06D;
   // UNICODE_TO_GBK[26292] := 16#7E8D;
   // UNICODE_TO_GBK[26293] := 16#C06E;
   // UNICODE_TO_GBK[26294] := 16#7E8E;
   // UNICODE_TO_GBK[26295] := 16#C06F;
   // UNICODE_TO_GBK[26296] := 16#7E8F;
   // UNICODE_TO_GBK[26297] := 16#C070;
   // UNICODE_TO_GBK[26298] := 16#7E90;
   // UNICODE_TO_GBK[26299] := 16#C071;
   // UNICODE_TO_GBK[26300] := 16#7E91;
   // UNICODE_TO_GBK[26301] := 16#C072;
   // UNICODE_TO_GBK[26302] := 16#7E92;
   // UNICODE_TO_GBK[26303] := 16#C073;
   // UNICODE_TO_GBK[26304] := 16#7E93;
   // UNICODE_TO_GBK[26305] := 16#C074;
   // UNICODE_TO_GBK[26306] := 16#7E94;
   // UNICODE_TO_GBK[26307] := 16#C075;
   // UNICODE_TO_GBK[26308] := 16#7E95;
   // UNICODE_TO_GBK[26309] := 16#C076;
   // UNICODE_TO_GBK[26310] := 16#7E96;
   // UNICODE_TO_GBK[26311] := 16#C077;
   // UNICODE_TO_GBK[26312] := 16#7E97;
   // UNICODE_TO_GBK[26313] := 16#C078;
   // UNICODE_TO_GBK[26314] := 16#7E98;
   // UNICODE_TO_GBK[26315] := 16#C079;
   // UNICODE_TO_GBK[26316] := 16#7E99;
   // UNICODE_TO_GBK[26317] := 16#C07A;
   // UNICODE_TO_GBK[26318] := 16#7E9A;
   // UNICODE_TO_GBK[26319] := 16#C07B;
   // UNICODE_TO_GBK[26320] := 16#7E9B;
   // UNICODE_TO_GBK[26321] := 16#F4EE;
   // UNICODE_TO_GBK[26322] := 16#7E9C;
   // UNICODE_TO_GBK[26323] := 16#C07C;
   // UNICODE_TO_GBK[26324] := 16#7E9D;
   // UNICODE_TO_GBK[26325] := 16#C07D;
   // UNICODE_TO_GBK[26326] := 16#7E9E;
   // UNICODE_TO_GBK[26327] := 16#C07E;
   // UNICODE_TO_GBK[26328] := 16#7E9F;
   // UNICODE_TO_GBK[26329] := 16#E6F9;
   // UNICODE_TO_GBK[26330] := 16#7EA0;
   // UNICODE_TO_GBK[26331] := 16#BEC0;
   // UNICODE_TO_GBK[26332] := 16#7EA1;
   // UNICODE_TO_GBK[26333] := 16#E6FA;
   // UNICODE_TO_GBK[26334] := 16#7EA2;
   // UNICODE_TO_GBK[26335] := 16#BAEC;
   // UNICODE_TO_GBK[26336] := 16#7EA3;
   // UNICODE_TO_GBK[26337] := 16#E6FB;
   // UNICODE_TO_GBK[26338] := 16#7EA4;
   // UNICODE_TO_GBK[26339] := 16#CFCB;
   // UNICODE_TO_GBK[26340] := 16#7EA5;
   // UNICODE_TO_GBK[26341] := 16#E6FC;
   // UNICODE_TO_GBK[26342] := 16#7EA6;
   // UNICODE_TO_GBK[26343] := 16#D4BC;
   // UNICODE_TO_GBK[26344] := 16#7EA7;
   // UNICODE_TO_GBK[26345] := 16#BCB6;
   // UNICODE_TO_GBK[26346] := 16#7EA8;
   // UNICODE_TO_GBK[26347] := 16#E6FD;
   // UNICODE_TO_GBK[26348] := 16#7EA9;
   // UNICODE_TO_GBK[26349] := 16#E6FE;
   // UNICODE_TO_GBK[26350] := 16#7EAA;
   // UNICODE_TO_GBK[26351] := 16#BCCD;
   // UNICODE_TO_GBK[26352] := 16#7EAB;
   // UNICODE_TO_GBK[26353] := 16#C8D2;
   // UNICODE_TO_GBK[26354] := 16#7EAC;
   // UNICODE_TO_GBK[26355] := 16#CEB3;
   // UNICODE_TO_GBK[26356] := 16#7EAD;
   // UNICODE_TO_GBK[26357] := 16#E7A1;
   // UNICODE_TO_GBK[26358] := 16#7EAE;
   // UNICODE_TO_GBK[26359] := 16#C080;
   // UNICODE_TO_GBK[26360] := 16#7EAF;
   // UNICODE_TO_GBK[26361] := 16#B4BF;
   // UNICODE_TO_GBK[26362] := 16#7EB0;
   // UNICODE_TO_GBK[26363] := 16#E7A2;
   // UNICODE_TO_GBK[26364] := 16#7EB1;
   // UNICODE_TO_GBK[26365] := 16#C9B4;
   // UNICODE_TO_GBK[26366] := 16#7EB2;
   // UNICODE_TO_GBK[26367] := 16#B8D9;
   // UNICODE_TO_GBK[26368] := 16#7EB3;
   // UNICODE_TO_GBK[26369] := 16#C4C9;
   // UNICODE_TO_GBK[26370] := 16#7EB4;
   // UNICODE_TO_GBK[26371] := 16#C081;
   // UNICODE_TO_GBK[26372] := 16#7EB5;
   // UNICODE_TO_GBK[26373] := 16#D7DD;
   // UNICODE_TO_GBK[26374] := 16#7EB6;
   // UNICODE_TO_GBK[26375] := 16#C2DA;
   // UNICODE_TO_GBK[26376] := 16#7EB7;
   // UNICODE_TO_GBK[26377] := 16#B7D7;
   // UNICODE_TO_GBK[26378] := 16#7EB8;
   // UNICODE_TO_GBK[26379] := 16#D6BD;
   // UNICODE_TO_GBK[26380] := 16#7EB9;
   // UNICODE_TO_GBK[26381] := 16#CEC6;
   // UNICODE_TO_GBK[26382] := 16#7EBA;
   // UNICODE_TO_GBK[26383] := 16#B7C4;
   // UNICODE_TO_GBK[26384] := 16#7EBB;
   // UNICODE_TO_GBK[26385] := 16#C082;
   // UNICODE_TO_GBK[26386] := 16#7EBC;
   // UNICODE_TO_GBK[26387] := 16#C083;
   // UNICODE_TO_GBK[26388] := 16#7EBD;
   // UNICODE_TO_GBK[26389] := 16#C5A6;
   // UNICODE_TO_GBK[26390] := 16#7EBE;
   // UNICODE_TO_GBK[26391] := 16#E7A3;
   // UNICODE_TO_GBK[26392] := 16#7EBF;
   // UNICODE_TO_GBK[26393] := 16#CFDF;
   // UNICODE_TO_GBK[26394] := 16#7EC0;
   // UNICODE_TO_GBK[26395] := 16#E7A4;
   // UNICODE_TO_GBK[26396] := 16#7EC1;
   // UNICODE_TO_GBK[26397] := 16#E7A5;
   // UNICODE_TO_GBK[26398] := 16#7EC2;
   // UNICODE_TO_GBK[26399] := 16#E7A6;
   // UNICODE_TO_GBK[26400] := 16#7EC3;
   // UNICODE_TO_GBK[26401] := 16#C1B7;
   // UNICODE_TO_GBK[26402] := 16#7EC4;
   // UNICODE_TO_GBK[26403] := 16#D7E9;
   // UNICODE_TO_GBK[26404] := 16#7EC5;
   // UNICODE_TO_GBK[26405] := 16#C9F0;
   // UNICODE_TO_GBK[26406] := 16#7EC6;
   // UNICODE_TO_GBK[26407] := 16#CFB8;
   // UNICODE_TO_GBK[26408] := 16#7EC7;
   // UNICODE_TO_GBK[26409] := 16#D6AF;
   // UNICODE_TO_GBK[26410] := 16#7EC8;
   // UNICODE_TO_GBK[26411] := 16#D6D5;
   // UNICODE_TO_GBK[26412] := 16#7EC9;
   // UNICODE_TO_GBK[26413] := 16#E7A7;
   // UNICODE_TO_GBK[26414] := 16#7ECA;
   // UNICODE_TO_GBK[26415] := 16#B0ED;
   // UNICODE_TO_GBK[26416] := 16#7ECB;
   // UNICODE_TO_GBK[26417] := 16#E7A8;
   // UNICODE_TO_GBK[26418] := 16#7ECC;
   // UNICODE_TO_GBK[26419] := 16#E7A9;
   // UNICODE_TO_GBK[26420] := 16#7ECD;
   // UNICODE_TO_GBK[26421] := 16#C9DC;
   // UNICODE_TO_GBK[26422] := 16#7ECE;
   // UNICODE_TO_GBK[26423] := 16#D2EF;
   // UNICODE_TO_GBK[26424] := 16#7ECF;
   // UNICODE_TO_GBK[26425] := 16#BEAD;
   // UNICODE_TO_GBK[26426] := 16#7ED0;
   // UNICODE_TO_GBK[26427] := 16#E7AA;
   // UNICODE_TO_GBK[26428] := 16#7ED1;
   // UNICODE_TO_GBK[26429] := 16#B0F3;
   // UNICODE_TO_GBK[26430] := 16#7ED2;
   // UNICODE_TO_GBK[26431] := 16#C8DE;
   // UNICODE_TO_GBK[26432] := 16#7ED3;
   // UNICODE_TO_GBK[26433] := 16#BDE1;
   // UNICODE_TO_GBK[26434] := 16#7ED4;
   // UNICODE_TO_GBK[26435] := 16#E7AB;
   // UNICODE_TO_GBK[26436] := 16#7ED5;
   // UNICODE_TO_GBK[26437] := 16#C8C6;
   // UNICODE_TO_GBK[26438] := 16#7ED6;
   // UNICODE_TO_GBK[26439] := 16#C084;
   // UNICODE_TO_GBK[26440] := 16#7ED7;
   // UNICODE_TO_GBK[26441] := 16#E7AC;
   // UNICODE_TO_GBK[26442] := 16#7ED8;
   // UNICODE_TO_GBK[26443] := 16#BBE6;
   // UNICODE_TO_GBK[26444] := 16#7ED9;
   // UNICODE_TO_GBK[26445] := 16#B8F8;
   // UNICODE_TO_GBK[26446] := 16#7EDA;
   // UNICODE_TO_GBK[26447] := 16#D1A4;
   // UNICODE_TO_GBK[26448] := 16#7EDB;
   // UNICODE_TO_GBK[26449] := 16#E7AD;
   // UNICODE_TO_GBK[26450] := 16#7EDC;
   // UNICODE_TO_GBK[26451] := 16#C2E7;
   // UNICODE_TO_GBK[26452] := 16#7EDD;
   // UNICODE_TO_GBK[26453] := 16#BEF8;
   // UNICODE_TO_GBK[26454] := 16#7EDE;
   // UNICODE_TO_GBK[26455] := 16#BDCA;
   // UNICODE_TO_GBK[26456] := 16#7EDF;
   // UNICODE_TO_GBK[26457] := 16#CDB3;
   // UNICODE_TO_GBK[26458] := 16#7EE0;
   // UNICODE_TO_GBK[26459] := 16#E7AE;
   // UNICODE_TO_GBK[26460] := 16#7EE1;
   // UNICODE_TO_GBK[26461] := 16#E7AF;
   // UNICODE_TO_GBK[26462] := 16#7EE2;
   // UNICODE_TO_GBK[26463] := 16#BEEE;
   // UNICODE_TO_GBK[26464] := 16#7EE3;
   // UNICODE_TO_GBK[26465] := 16#D0E5;
   // UNICODE_TO_GBK[26466] := 16#7EE4;
   // UNICODE_TO_GBK[26467] := 16#C085;
   // UNICODE_TO_GBK[26468] := 16#7EE5;
   // UNICODE_TO_GBK[26469] := 16#CBE7;
   // UNICODE_TO_GBK[26470] := 16#7EE6;
   // UNICODE_TO_GBK[26471] := 16#CCD0;
   // UNICODE_TO_GBK[26472] := 16#7EE7;
   // UNICODE_TO_GBK[26473] := 16#BCCC;
   // UNICODE_TO_GBK[26474] := 16#7EE8;
   // UNICODE_TO_GBK[26475] := 16#E7B0;
   // UNICODE_TO_GBK[26476] := 16#7EE9;
   // UNICODE_TO_GBK[26477] := 16#BCA8;
   // UNICODE_TO_GBK[26478] := 16#7EEA;
   // UNICODE_TO_GBK[26479] := 16#D0F7;
   // UNICODE_TO_GBK[26480] := 16#7EEB;
   // UNICODE_TO_GBK[26481] := 16#E7B1;
   // UNICODE_TO_GBK[26482] := 16#7EEC;
   // UNICODE_TO_GBK[26483] := 16#C086;
   // UNICODE_TO_GBK[26484] := 16#7EED;
   // UNICODE_TO_GBK[26485] := 16#D0F8;
   // UNICODE_TO_GBK[26486] := 16#7EEE;
   // UNICODE_TO_GBK[26487] := 16#E7B2;
   // UNICODE_TO_GBK[26488] := 16#7EEF;
   // UNICODE_TO_GBK[26489] := 16#E7B3;
   // UNICODE_TO_GBK[26490] := 16#7EF0;
   // UNICODE_TO_GBK[26491] := 16#B4C2;
   // UNICODE_TO_GBK[26492] := 16#7EF1;
   // UNICODE_TO_GBK[26493] := 16#E7B4;
   // UNICODE_TO_GBK[26494] := 16#7EF2;
   // UNICODE_TO_GBK[26495] := 16#E7B5;
   // UNICODE_TO_GBK[26496] := 16#7EF3;
   // UNICODE_TO_GBK[26497] := 16#C9FE;
   // UNICODE_TO_GBK[26498] := 16#7EF4;
   // UNICODE_TO_GBK[26499] := 16#CEAC;
   // UNICODE_TO_GBK[26500] := 16#7EF5;
   // UNICODE_TO_GBK[26501] := 16#C3E0;
   // UNICODE_TO_GBK[26502] := 16#7EF6;
   // UNICODE_TO_GBK[26503] := 16#E7B7;
   // UNICODE_TO_GBK[26504] := 16#7EF7;
   // UNICODE_TO_GBK[26505] := 16#B1C1;
   // UNICODE_TO_GBK[26506] := 16#7EF8;
   // UNICODE_TO_GBK[26507] := 16#B3F1;
   // UNICODE_TO_GBK[26508] := 16#7EF9;
   // UNICODE_TO_GBK[26509] := 16#C087;
   // UNICODE_TO_GBK[26510] := 16#7EFA;
   // UNICODE_TO_GBK[26511] := 16#E7B8;
   // UNICODE_TO_GBK[26512] := 16#7EFB;
   // UNICODE_TO_GBK[26513] := 16#E7B9;
   // UNICODE_TO_GBK[26514] := 16#7EFC;
   // UNICODE_TO_GBK[26515] := 16#D7DB;
   // UNICODE_TO_GBK[26516] := 16#7EFD;
   // UNICODE_TO_GBK[26517] := 16#D5C0;
   // UNICODE_TO_GBK[26518] := 16#7EFE;
   // UNICODE_TO_GBK[26519] := 16#E7BA;
   // UNICODE_TO_GBK[26520] := 16#7EFF;
   // UNICODE_TO_GBK[26521] := 16#C2CC;
   // UNICODE_TO_GBK[26522] := 16#7F00;
   // UNICODE_TO_GBK[26523] := 16#D7BA;
   // UNICODE_TO_GBK[26524] := 16#7F01;
   // UNICODE_TO_GBK[26525] := 16#E7BB;
   // UNICODE_TO_GBK[26526] := 16#7F02;
   // UNICODE_TO_GBK[26527] := 16#E7BC;
   // UNICODE_TO_GBK[26528] := 16#7F03;
   // UNICODE_TO_GBK[26529] := 16#E7BD;
   // UNICODE_TO_GBK[26530] := 16#7F04;
   // UNICODE_TO_GBK[26531] := 16#BCEA;
   // UNICODE_TO_GBK[26532] := 16#7F05;
   // UNICODE_TO_GBK[26533] := 16#C3E5;
   // UNICODE_TO_GBK[26534] := 16#7F06;
   // UNICODE_TO_GBK[26535] := 16#C0C2;
   // UNICODE_TO_GBK[26536] := 16#7F07;
   // UNICODE_TO_GBK[26537] := 16#E7BE;
   // UNICODE_TO_GBK[26538] := 16#7F08;
   // UNICODE_TO_GBK[26539] := 16#E7BF;
   // UNICODE_TO_GBK[26540] := 16#7F09;
   // UNICODE_TO_GBK[26541] := 16#BCA9;
   // UNICODE_TO_GBK[26542] := 16#7F0A;
   // UNICODE_TO_GBK[26543] := 16#C088;
   // UNICODE_TO_GBK[26544] := 16#7F0B;
   // UNICODE_TO_GBK[26545] := 16#E7C0;
   // UNICODE_TO_GBK[26546] := 16#7F0C;
   // UNICODE_TO_GBK[26547] := 16#E7C1;
   // UNICODE_TO_GBK[26548] := 16#7F0D;
   // UNICODE_TO_GBK[26549] := 16#E7B6;
   // UNICODE_TO_GBK[26550] := 16#7F0E;
   // UNICODE_TO_GBK[26551] := 16#B6D0;
   // UNICODE_TO_GBK[26552] := 16#7F0F;
   // UNICODE_TO_GBK[26553] := 16#E7C2;
   // UNICODE_TO_GBK[26554] := 16#7F10;
   // UNICODE_TO_GBK[26555] := 16#C089;
   // UNICODE_TO_GBK[26556] := 16#7F11;
   // UNICODE_TO_GBK[26557] := 16#E7C3;
   // UNICODE_TO_GBK[26558] := 16#7F12;
   // UNICODE_TO_GBK[26559] := 16#E7C4;
   // UNICODE_TO_GBK[26560] := 16#7F13;
   // UNICODE_TO_GBK[26561] := 16#BBBA;
   // UNICODE_TO_GBK[26562] := 16#7F14;
   // UNICODE_TO_GBK[26563] := 16#B5DE;
   // UNICODE_TO_GBK[26564] := 16#7F15;
   // UNICODE_TO_GBK[26565] := 16#C2C6;
   // UNICODE_TO_GBK[26566] := 16#7F16;
   // UNICODE_TO_GBK[26567] := 16#B1E0;
   // UNICODE_TO_GBK[26568] := 16#7F17;
   // UNICODE_TO_GBK[26569] := 16#E7C5;
   // UNICODE_TO_GBK[26570] := 16#7F18;
   // UNICODE_TO_GBK[26571] := 16#D4B5;
   // UNICODE_TO_GBK[26572] := 16#7F19;
   // UNICODE_TO_GBK[26573] := 16#E7C6;
   // UNICODE_TO_GBK[26574] := 16#7F1A;
   // UNICODE_TO_GBK[26575] := 16#B8BF;
   // UNICODE_TO_GBK[26576] := 16#7F1B;
   // UNICODE_TO_GBK[26577] := 16#E7C8;
   // UNICODE_TO_GBK[26578] := 16#7F1C;
   // UNICODE_TO_GBK[26579] := 16#E7C7;
   // UNICODE_TO_GBK[26580] := 16#7F1D;
   // UNICODE_TO_GBK[26581] := 16#B7EC;
   // UNICODE_TO_GBK[26582] := 16#7F1E;
   // UNICODE_TO_GBK[26583] := 16#C08A;
   // UNICODE_TO_GBK[26584] := 16#7F1F;
   // UNICODE_TO_GBK[26585] := 16#E7C9;
   // UNICODE_TO_GBK[26586] := 16#7F20;
   // UNICODE_TO_GBK[26587] := 16#B2F8;
   // UNICODE_TO_GBK[26588] := 16#7F21;
   // UNICODE_TO_GBK[26589] := 16#E7CA;
   // UNICODE_TO_GBK[26590] := 16#7F22;
   // UNICODE_TO_GBK[26591] := 16#E7CB;
   // UNICODE_TO_GBK[26592] := 16#7F23;
   // UNICODE_TO_GBK[26593] := 16#E7CC;
   // UNICODE_TO_GBK[26594] := 16#7F24;
   // UNICODE_TO_GBK[26595] := 16#E7CD;
   // UNICODE_TO_GBK[26596] := 16#7F25;
   // UNICODE_TO_GBK[26597] := 16#E7CE;
   // UNICODE_TO_GBK[26598] := 16#7F26;
   // UNICODE_TO_GBK[26599] := 16#E7CF;
   // UNICODE_TO_GBK[26600] := 16#7F27;
   // UNICODE_TO_GBK[26601] := 16#E7D0;
   // UNICODE_TO_GBK[26602] := 16#7F28;
   // UNICODE_TO_GBK[26603] := 16#D3A7;
   // UNICODE_TO_GBK[26604] := 16#7F29;
   // UNICODE_TO_GBK[26605] := 16#CBF5;
   // UNICODE_TO_GBK[26606] := 16#7F2A;
   // UNICODE_TO_GBK[26607] := 16#E7D1;
   // UNICODE_TO_GBK[26608] := 16#7F2B;
   // UNICODE_TO_GBK[26609] := 16#E7D2;
   // UNICODE_TO_GBK[26610] := 16#7F2C;
   // UNICODE_TO_GBK[26611] := 16#E7D3;
   // UNICODE_TO_GBK[26612] := 16#7F2D;
   // UNICODE_TO_GBK[26613] := 16#E7D4;
   // UNICODE_TO_GBK[26614] := 16#7F2E;
   // UNICODE_TO_GBK[26615] := 16#C9C9;
   // UNICODE_TO_GBK[26616] := 16#7F2F;
   // UNICODE_TO_GBK[26617] := 16#E7D5;
   // UNICODE_TO_GBK[26618] := 16#7F30;
   // UNICODE_TO_GBK[26619] := 16#E7D6;
   // UNICODE_TO_GBK[26620] := 16#7F31;
   // UNICODE_TO_GBK[26621] := 16#E7D7;
   // UNICODE_TO_GBK[26622] := 16#7F32;
   // UNICODE_TO_GBK[26623] := 16#E7D8;
   // UNICODE_TO_GBK[26624] := 16#7F33;
   // UNICODE_TO_GBK[26625] := 16#E7D9;
   // UNICODE_TO_GBK[26626] := 16#7F34;
   // UNICODE_TO_GBK[26627] := 16#BDC9;
   // UNICODE_TO_GBK[26628] := 16#7F35;
   // UNICODE_TO_GBK[26629] := 16#E7DA;
   // UNICODE_TO_GBK[26630] := 16#7F36;
   // UNICODE_TO_GBK[26631] := 16#F3BE;
   // UNICODE_TO_GBK[26632] := 16#7F37;
   // UNICODE_TO_GBK[26633] := 16#C08B;
   // UNICODE_TO_GBK[26634] := 16#7F38;
   // UNICODE_TO_GBK[26635] := 16#B8D7;
   // UNICODE_TO_GBK[26636] := 16#7F39;
   // UNICODE_TO_GBK[26637] := 16#C08C;
   // UNICODE_TO_GBK[26638] := 16#7F3A;
   // UNICODE_TO_GBK[26639] := 16#C8B1;
   // UNICODE_TO_GBK[26640] := 16#7F3B;
   // UNICODE_TO_GBK[26641] := 16#C08D;
   // UNICODE_TO_GBK[26642] := 16#7F3C;
   // UNICODE_TO_GBK[26643] := 16#C08E;
   // UNICODE_TO_GBK[26644] := 16#7F3D;
   // UNICODE_TO_GBK[26645] := 16#C08F;
   // UNICODE_TO_GBK[26646] := 16#7F3E;
   // UNICODE_TO_GBK[26647] := 16#C090;
   // UNICODE_TO_GBK[26648] := 16#7F3F;
   // UNICODE_TO_GBK[26649] := 16#C091;
   // UNICODE_TO_GBK[26650] := 16#7F40;
   // UNICODE_TO_GBK[26651] := 16#C092;
   // UNICODE_TO_GBK[26652] := 16#7F41;
   // UNICODE_TO_GBK[26653] := 16#C093;
   // UNICODE_TO_GBK[26654] := 16#7F42;
   // UNICODE_TO_GBK[26655] := 16#F3BF;
   // UNICODE_TO_GBK[26656] := 16#7F43;
   // UNICODE_TO_GBK[26657] := 16#C094;
   // UNICODE_TO_GBK[26658] := 16#7F44;
   // UNICODE_TO_GBK[26659] := 16#F3C0;
   // UNICODE_TO_GBK[26660] := 16#7F45;
   // UNICODE_TO_GBK[26661] := 16#F3C1;
   // UNICODE_TO_GBK[26662] := 16#7F46;
   // UNICODE_TO_GBK[26663] := 16#C095;
   // UNICODE_TO_GBK[26664] := 16#7F47;
   // UNICODE_TO_GBK[26665] := 16#C096;
   // UNICODE_TO_GBK[26666] := 16#7F48;
   // UNICODE_TO_GBK[26667] := 16#C097;
   // UNICODE_TO_GBK[26668] := 16#7F49;
   // UNICODE_TO_GBK[26669] := 16#C098;
   // UNICODE_TO_GBK[26670] := 16#7F4A;
   // UNICODE_TO_GBK[26671] := 16#C099;
   // UNICODE_TO_GBK[26672] := 16#7F4B;
   // UNICODE_TO_GBK[26673] := 16#C09A;
   // UNICODE_TO_GBK[26674] := 16#7F4C;
   // UNICODE_TO_GBK[26675] := 16#C09B;
   // UNICODE_TO_GBK[26676] := 16#7F4D;
   // UNICODE_TO_GBK[26677] := 16#C09C;
   // UNICODE_TO_GBK[26678] := 16#7F4E;
   // UNICODE_TO_GBK[26679] := 16#C09D;
   // UNICODE_TO_GBK[26680] := 16#7F4F;
   // UNICODE_TO_GBK[26681] := 16#C09E;
   // UNICODE_TO_GBK[26682] := 16#7F50;
   // UNICODE_TO_GBK[26683] := 16#B9DE;
   // UNICODE_TO_GBK[26684] := 16#7F51;
   // UNICODE_TO_GBK[26685] := 16#CDF8;
   // UNICODE_TO_GBK[26686] := 16#7F52;
   // UNICODE_TO_GBK[26687] := 16#C09F;
   // UNICODE_TO_GBK[26688] := 16#7F53;
   // UNICODE_TO_GBK[26689] := 16#C0A0;
   // UNICODE_TO_GBK[26690] := 16#7F54;
   // UNICODE_TO_GBK[26691] := 16#D8E8;
   // UNICODE_TO_GBK[26692] := 16#7F55;
   // UNICODE_TO_GBK[26693] := 16#BAB1;
   // UNICODE_TO_GBK[26694] := 16#7F56;
   // UNICODE_TO_GBK[26695] := 16#C140;
   // UNICODE_TO_GBK[26696] := 16#7F57;
   // UNICODE_TO_GBK[26697] := 16#C2DE;
   // UNICODE_TO_GBK[26698] := 16#7F58;
   // UNICODE_TO_GBK[26699] := 16#EEB7;
   // UNICODE_TO_GBK[26700] := 16#7F59;
   // UNICODE_TO_GBK[26701] := 16#C141;
   // UNICODE_TO_GBK[26702] := 16#7F5A;
   // UNICODE_TO_GBK[26703] := 16#B7A3;
   // UNICODE_TO_GBK[26704] := 16#7F5B;
   // UNICODE_TO_GBK[26705] := 16#C142;
   // UNICODE_TO_GBK[26706] := 16#7F5C;
   // UNICODE_TO_GBK[26707] := 16#C143;
   // UNICODE_TO_GBK[26708] := 16#7F5D;
   // UNICODE_TO_GBK[26709] := 16#C144;
   // UNICODE_TO_GBK[26710] := 16#7F5E;
   // UNICODE_TO_GBK[26711] := 16#C145;
   // UNICODE_TO_GBK[26712] := 16#7F5F;
   // UNICODE_TO_GBK[26713] := 16#EEB9;
   // UNICODE_TO_GBK[26714] := 16#7F60;
   // UNICODE_TO_GBK[26715] := 16#C146;
   // UNICODE_TO_GBK[26716] := 16#7F61;
   // UNICODE_TO_GBK[26717] := 16#EEB8;
   // UNICODE_TO_GBK[26718] := 16#7F62;
   // UNICODE_TO_GBK[26719] := 16#B0D5;
   // UNICODE_TO_GBK[26720] := 16#7F63;
   // UNICODE_TO_GBK[26721] := 16#C147;
   // UNICODE_TO_GBK[26722] := 16#7F64;
   // UNICODE_TO_GBK[26723] := 16#C148;
   // UNICODE_TO_GBK[26724] := 16#7F65;
   // UNICODE_TO_GBK[26725] := 16#C149;
   // UNICODE_TO_GBK[26726] := 16#7F66;
   // UNICODE_TO_GBK[26727] := 16#C14A;
   // UNICODE_TO_GBK[26728] := 16#7F67;
   // UNICODE_TO_GBK[26729] := 16#C14B;
   // UNICODE_TO_GBK[26730] := 16#7F68;
   // UNICODE_TO_GBK[26731] := 16#EEBB;
   // UNICODE_TO_GBK[26732] := 16#7F69;
   // UNICODE_TO_GBK[26733] := 16#D5D6;
   // UNICODE_TO_GBK[26734] := 16#7F6A;
   // UNICODE_TO_GBK[26735] := 16#D7EF;
   // UNICODE_TO_GBK[26736] := 16#7F6B;
   // UNICODE_TO_GBK[26737] := 16#C14C;
   // UNICODE_TO_GBK[26738] := 16#7F6C;
   // UNICODE_TO_GBK[26739] := 16#C14D;
   // UNICODE_TO_GBK[26740] := 16#7F6D;
   // UNICODE_TO_GBK[26741] := 16#C14E;
   // UNICODE_TO_GBK[26742] := 16#7F6E;
   // UNICODE_TO_GBK[26743] := 16#D6C3;
   // UNICODE_TO_GBK[26744] := 16#7F6F;
   // UNICODE_TO_GBK[26745] := 16#C14F;
   // UNICODE_TO_GBK[26746] := 16#7F70;
   // UNICODE_TO_GBK[26747] := 16#C150;
   // UNICODE_TO_GBK[26748] := 16#7F71;
   // UNICODE_TO_GBK[26749] := 16#EEBD;
   // UNICODE_TO_GBK[26750] := 16#7F72;
   // UNICODE_TO_GBK[26751] := 16#CAF0;
   // UNICODE_TO_GBK[26752] := 16#7F73;
   // UNICODE_TO_GBK[26753] := 16#C151;
   // UNICODE_TO_GBK[26754] := 16#7F74;
   // UNICODE_TO_GBK[26755] := 16#EEBC;
   // UNICODE_TO_GBK[26756] := 16#7F75;
   // UNICODE_TO_GBK[26757] := 16#C152;
   // UNICODE_TO_GBK[26758] := 16#7F76;
   // UNICODE_TO_GBK[26759] := 16#C153;
   // UNICODE_TO_GBK[26760] := 16#7F77;
   // UNICODE_TO_GBK[26761] := 16#C154;
   // UNICODE_TO_GBK[26762] := 16#7F78;
   // UNICODE_TO_GBK[26763] := 16#C155;
   // UNICODE_TO_GBK[26764] := 16#7F79;
   // UNICODE_TO_GBK[26765] := 16#EEBE;
   // UNICODE_TO_GBK[26766] := 16#7F7A;
   // UNICODE_TO_GBK[26767] := 16#C156;
   // UNICODE_TO_GBK[26768] := 16#7F7B;
   // UNICODE_TO_GBK[26769] := 16#C157;
   // UNICODE_TO_GBK[26770] := 16#7F7C;
   // UNICODE_TO_GBK[26771] := 16#C158;
   // UNICODE_TO_GBK[26772] := 16#7F7D;
   // UNICODE_TO_GBK[26773] := 16#C159;
   // UNICODE_TO_GBK[26774] := 16#7F7E;
   // UNICODE_TO_GBK[26775] := 16#EEC0;
   // UNICODE_TO_GBK[26776] := 16#7F7F;
   // UNICODE_TO_GBK[26777] := 16#C15A;
   // UNICODE_TO_GBK[26778] := 16#7F80;
   // UNICODE_TO_GBK[26779] := 16#C15B;
   // UNICODE_TO_GBK[26780] := 16#7F81;
   // UNICODE_TO_GBK[26781] := 16#EEBF;
   // UNICODE_TO_GBK[26782] := 16#7F82;
   // UNICODE_TO_GBK[26783] := 16#C15C;
   // UNICODE_TO_GBK[26784] := 16#7F83;
   // UNICODE_TO_GBK[26785] := 16#C15D;
   // UNICODE_TO_GBK[26786] := 16#7F84;
   // UNICODE_TO_GBK[26787] := 16#C15E;
   // UNICODE_TO_GBK[26788] := 16#7F85;
   // UNICODE_TO_GBK[26789] := 16#C15F;
   // UNICODE_TO_GBK[26790] := 16#7F86;
   // UNICODE_TO_GBK[26791] := 16#C160;
   // UNICODE_TO_GBK[26792] := 16#7F87;
   // UNICODE_TO_GBK[26793] := 16#C161;
   // UNICODE_TO_GBK[26794] := 16#7F88;
   // UNICODE_TO_GBK[26795] := 16#C162;
   // UNICODE_TO_GBK[26796] := 16#7F89;
   // UNICODE_TO_GBK[26797] := 16#C163;
   // UNICODE_TO_GBK[26798] := 16#7F8A;
   // UNICODE_TO_GBK[26799] := 16#D1F2;
   // UNICODE_TO_GBK[26800] := 16#7F8B;
   // UNICODE_TO_GBK[26801] := 16#C164;
   // UNICODE_TO_GBK[26802] := 16#7F8C;
   // UNICODE_TO_GBK[26803] := 16#C7BC;
   // UNICODE_TO_GBK[26804] := 16#7F8D;
   // UNICODE_TO_GBK[26805] := 16#C165;
   // UNICODE_TO_GBK[26806] := 16#7F8E;
   // UNICODE_TO_GBK[26807] := 16#C3C0;
   // UNICODE_TO_GBK[26808] := 16#7F8F;
   // UNICODE_TO_GBK[26809] := 16#C166;
   // UNICODE_TO_GBK[26810] := 16#7F90;
   // UNICODE_TO_GBK[26811] := 16#C167;
   // UNICODE_TO_GBK[26812] := 16#7F91;
   // UNICODE_TO_GBK[26813] := 16#C168;
   // UNICODE_TO_GBK[26814] := 16#7F92;
   // UNICODE_TO_GBK[26815] := 16#C169;
   // UNICODE_TO_GBK[26816] := 16#7F93;
   // UNICODE_TO_GBK[26817] := 16#C16A;
   // UNICODE_TO_GBK[26818] := 16#7F94;
   // UNICODE_TO_GBK[26819] := 16#B8E1;
   // UNICODE_TO_GBK[26820] := 16#7F95;
   // UNICODE_TO_GBK[26821] := 16#C16B;
   // UNICODE_TO_GBK[26822] := 16#7F96;
   // UNICODE_TO_GBK[26823] := 16#C16C;
   // UNICODE_TO_GBK[26824] := 16#7F97;
   // UNICODE_TO_GBK[26825] := 16#C16D;
   // UNICODE_TO_GBK[26826] := 16#7F98;
   // UNICODE_TO_GBK[26827] := 16#C16E;
   // UNICODE_TO_GBK[26828] := 16#7F99;
   // UNICODE_TO_GBK[26829] := 16#C16F;
   // UNICODE_TO_GBK[26830] := 16#7F9A;
   // UNICODE_TO_GBK[26831] := 16#C1E7;
   // UNICODE_TO_GBK[26832] := 16#7F9B;
   // UNICODE_TO_GBK[26833] := 16#C170;
   // UNICODE_TO_GBK[26834] := 16#7F9C;
   // UNICODE_TO_GBK[26835] := 16#C171;
   // UNICODE_TO_GBK[26836] := 16#7F9D;
   // UNICODE_TO_GBK[26837] := 16#F4C6;
   // UNICODE_TO_GBK[26838] := 16#7F9E;
   // UNICODE_TO_GBK[26839] := 16#D0DF;
   // UNICODE_TO_GBK[26840] := 16#7F9F;
   // UNICODE_TO_GBK[26841] := 16#F4C7;
   // UNICODE_TO_GBK[26842] := 16#7FA0;
   // UNICODE_TO_GBK[26843] := 16#C172;
   // UNICODE_TO_GBK[26844] := 16#7FA1;
   // UNICODE_TO_GBK[26845] := 16#CFDB;
   // UNICODE_TO_GBK[26846] := 16#7FA2;
   // UNICODE_TO_GBK[26847] := 16#C173;
   // UNICODE_TO_GBK[26848] := 16#7FA3;
   // UNICODE_TO_GBK[26849] := 16#C174;
   // UNICODE_TO_GBK[26850] := 16#7FA4;
   // UNICODE_TO_GBK[26851] := 16#C8BA;
   // UNICODE_TO_GBK[26852] := 16#7FA5;
   // UNICODE_TO_GBK[26853] := 16#C175;
   // UNICODE_TO_GBK[26854] := 16#7FA6;
   // UNICODE_TO_GBK[26855] := 16#C176;
   // UNICODE_TO_GBK[26856] := 16#7FA7;
   // UNICODE_TO_GBK[26857] := 16#F4C8;
   // UNICODE_TO_GBK[26858] := 16#7FA8;
   // UNICODE_TO_GBK[26859] := 16#C177;
   // UNICODE_TO_GBK[26860] := 16#7FA9;
   // UNICODE_TO_GBK[26861] := 16#C178;
   // UNICODE_TO_GBK[26862] := 16#7FAA;
   // UNICODE_TO_GBK[26863] := 16#C179;
   // UNICODE_TO_GBK[26864] := 16#7FAB;
   // UNICODE_TO_GBK[26865] := 16#C17A;
   // UNICODE_TO_GBK[26866] := 16#7FAC;
   // UNICODE_TO_GBK[26867] := 16#C17B;
   // UNICODE_TO_GBK[26868] := 16#7FAD;
   // UNICODE_TO_GBK[26869] := 16#C17C;
   // UNICODE_TO_GBK[26870] := 16#7FAE;
   // UNICODE_TO_GBK[26871] := 16#C17D;
   // UNICODE_TO_GBK[26872] := 16#7FAF;
   // UNICODE_TO_GBK[26873] := 16#F4C9;
   // UNICODE_TO_GBK[26874] := 16#7FB0;
   // UNICODE_TO_GBK[26875] := 16#F4CA;
   // UNICODE_TO_GBK[26876] := 16#7FB1;
   // UNICODE_TO_GBK[26877] := 16#C17E;
   // UNICODE_TO_GBK[26878] := 16#7FB2;
   // UNICODE_TO_GBK[26879] := 16#F4CB;
   // UNICODE_TO_GBK[26880] := 16#7FB3;
   // UNICODE_TO_GBK[26881] := 16#C180;
   // UNICODE_TO_GBK[26882] := 16#7FB4;
   // UNICODE_TO_GBK[26883] := 16#C181;
   // UNICODE_TO_GBK[26884] := 16#7FB5;
   // UNICODE_TO_GBK[26885] := 16#C182;
   // UNICODE_TO_GBK[26886] := 16#7FB6;
   // UNICODE_TO_GBK[26887] := 16#C183;
   // UNICODE_TO_GBK[26888] := 16#7FB7;
   // UNICODE_TO_GBK[26889] := 16#C184;
   // UNICODE_TO_GBK[26890] := 16#7FB8;
   // UNICODE_TO_GBK[26891] := 16#D9FA;
   // UNICODE_TO_GBK[26892] := 16#7FB9;
   // UNICODE_TO_GBK[26893] := 16#B8FE;
   // UNICODE_TO_GBK[26894] := 16#7FBA;
   // UNICODE_TO_GBK[26895] := 16#C185;
   // UNICODE_TO_GBK[26896] := 16#7FBB;
   // UNICODE_TO_GBK[26897] := 16#C186;
   // UNICODE_TO_GBK[26898] := 16#7FBC;
   // UNICODE_TO_GBK[26899] := 16#E5F1;
   // UNICODE_TO_GBK[26900] := 16#7FBD;
   // UNICODE_TO_GBK[26901] := 16#D3F0;
   // UNICODE_TO_GBK[26902] := 16#7FBE;
   // UNICODE_TO_GBK[26903] := 16#C187;
   // UNICODE_TO_GBK[26904] := 16#7FBF;
   // UNICODE_TO_GBK[26905] := 16#F4E0;
   // UNICODE_TO_GBK[26906] := 16#7FC0;
   // UNICODE_TO_GBK[26907] := 16#C188;
   // UNICODE_TO_GBK[26908] := 16#7FC1;
   // UNICODE_TO_GBK[26909] := 16#CECC;
   // UNICODE_TO_GBK[26910] := 16#7FC2;
   // UNICODE_TO_GBK[26911] := 16#C189;
   // UNICODE_TO_GBK[26912] := 16#7FC3;
   // UNICODE_TO_GBK[26913] := 16#C18A;
   // UNICODE_TO_GBK[26914] := 16#7FC4;
   // UNICODE_TO_GBK[26915] := 16#C18B;
   // UNICODE_TO_GBK[26916] := 16#7FC5;
   // UNICODE_TO_GBK[26917] := 16#B3E1;
   // UNICODE_TO_GBK[26918] := 16#7FC6;
   // UNICODE_TO_GBK[26919] := 16#C18C;
   // UNICODE_TO_GBK[26920] := 16#7FC7;
   // UNICODE_TO_GBK[26921] := 16#C18D;
   // UNICODE_TO_GBK[26922] := 16#7FC8;
   // UNICODE_TO_GBK[26923] := 16#C18E;
   // UNICODE_TO_GBK[26924] := 16#7FC9;
   // UNICODE_TO_GBK[26925] := 16#C18F;
   // UNICODE_TO_GBK[26926] := 16#7FCA;
   // UNICODE_TO_GBK[26927] := 16#F1B4;
   // UNICODE_TO_GBK[26928] := 16#7FCB;
   // UNICODE_TO_GBK[26929] := 16#C190;
   // UNICODE_TO_GBK[26930] := 16#7FCC;
   // UNICODE_TO_GBK[26931] := 16#D2EE;
   // UNICODE_TO_GBK[26932] := 16#7FCD;
   // UNICODE_TO_GBK[26933] := 16#C191;
   // UNICODE_TO_GBK[26934] := 16#7FCE;
   // UNICODE_TO_GBK[26935] := 16#F4E1;
   // UNICODE_TO_GBK[26936] := 16#7FCF;
   // UNICODE_TO_GBK[26937] := 16#C192;
   // UNICODE_TO_GBK[26938] := 16#7FD0;
   // UNICODE_TO_GBK[26939] := 16#C193;
   // UNICODE_TO_GBK[26940] := 16#7FD1;
   // UNICODE_TO_GBK[26941] := 16#C194;
   // UNICODE_TO_GBK[26942] := 16#7FD2;
   // UNICODE_TO_GBK[26943] := 16#C195;
   // UNICODE_TO_GBK[26944] := 16#7FD3;
   // UNICODE_TO_GBK[26945] := 16#C196;
   // UNICODE_TO_GBK[26946] := 16#7FD4;
   // UNICODE_TO_GBK[26947] := 16#CFE8;
   // UNICODE_TO_GBK[26948] := 16#7FD5;
   // UNICODE_TO_GBK[26949] := 16#F4E2;
   // UNICODE_TO_GBK[26950] := 16#7FD6;
   // UNICODE_TO_GBK[26951] := 16#C197;
   // UNICODE_TO_GBK[26952] := 16#7FD7;
   // UNICODE_TO_GBK[26953] := 16#C198;
   // UNICODE_TO_GBK[26954] := 16#7FD8;
   // UNICODE_TO_GBK[26955] := 16#C7CC;
   // UNICODE_TO_GBK[26956] := 16#7FD9;
   // UNICODE_TO_GBK[26957] := 16#C199;
   // UNICODE_TO_GBK[26958] := 16#7FDA;
   // UNICODE_TO_GBK[26959] := 16#C19A;
   // UNICODE_TO_GBK[26960] := 16#7FDB;
   // UNICODE_TO_GBK[26961] := 16#C19B;
   // UNICODE_TO_GBK[26962] := 16#7FDC;
   // UNICODE_TO_GBK[26963] := 16#C19C;
   // UNICODE_TO_GBK[26964] := 16#7FDD;
   // UNICODE_TO_GBK[26965] := 16#C19D;
   // UNICODE_TO_GBK[26966] := 16#7FDE;
   // UNICODE_TO_GBK[26967] := 16#C19E;
   // UNICODE_TO_GBK[26968] := 16#7FDF;
   // UNICODE_TO_GBK[26969] := 16#B5D4;
   // UNICODE_TO_GBK[26970] := 16#7FE0;
   // UNICODE_TO_GBK[26971] := 16#B4E4;
   // UNICODE_TO_GBK[26972] := 16#7FE1;
   // UNICODE_TO_GBK[26973] := 16#F4E4;
   // UNICODE_TO_GBK[26974] := 16#7FE2;
   // UNICODE_TO_GBK[26975] := 16#C19F;
   // UNICODE_TO_GBK[26976] := 16#7FE3;
   // UNICODE_TO_GBK[26977] := 16#C1A0;
   // UNICODE_TO_GBK[26978] := 16#7FE4;
   // UNICODE_TO_GBK[26979] := 16#C240;
   // UNICODE_TO_GBK[26980] := 16#7FE5;
   // UNICODE_TO_GBK[26981] := 16#F4E3;
   // UNICODE_TO_GBK[26982] := 16#7FE6;
   // UNICODE_TO_GBK[26983] := 16#F4E5;
   // UNICODE_TO_GBK[26984] := 16#7FE7;
   // UNICODE_TO_GBK[26985] := 16#C241;
   // UNICODE_TO_GBK[26986] := 16#7FE8;
   // UNICODE_TO_GBK[26987] := 16#C242;
   // UNICODE_TO_GBK[26988] := 16#7FE9;
   // UNICODE_TO_GBK[26989] := 16#F4E6;
   // UNICODE_TO_GBK[26990] := 16#7FEA;
   // UNICODE_TO_GBK[26991] := 16#C243;
   // UNICODE_TO_GBK[26992] := 16#7FEB;
   // UNICODE_TO_GBK[26993] := 16#C244;
   // UNICODE_TO_GBK[26994] := 16#7FEC;
   // UNICODE_TO_GBK[26995] := 16#C245;
   // UNICODE_TO_GBK[26996] := 16#7FED;
   // UNICODE_TO_GBK[26997] := 16#C246;
   // UNICODE_TO_GBK[26998] := 16#7FEE;
   // UNICODE_TO_GBK[26999] := 16#F4E7;
   // UNICODE_TO_GBK[27000] := 16#7FEF;
   // UNICODE_TO_GBK[27001] := 16#C247;
   // UNICODE_TO_GBK[27002] := 16#7FF0;
   // UNICODE_TO_GBK[27003] := 16#BAB2;
   // UNICODE_TO_GBK[27004] := 16#7FF1;
   // UNICODE_TO_GBK[27005] := 16#B0BF;
   // UNICODE_TO_GBK[27006] := 16#7FF2;
   // UNICODE_TO_GBK[27007] := 16#C248;
   // UNICODE_TO_GBK[27008] := 16#7FF3;
   // UNICODE_TO_GBK[27009] := 16#F4E8;
   // UNICODE_TO_GBK[27010] := 16#7FF4;
   // UNICODE_TO_GBK[27011] := 16#C249;
   // UNICODE_TO_GBK[27012] := 16#7FF5;
   // UNICODE_TO_GBK[27013] := 16#C24A;
   // UNICODE_TO_GBK[27014] := 16#7FF6;
   // UNICODE_TO_GBK[27015] := 16#C24B;
   // UNICODE_TO_GBK[27016] := 16#7FF7;
   // UNICODE_TO_GBK[27017] := 16#C24C;
   // UNICODE_TO_GBK[27018] := 16#7FF8;
   // UNICODE_TO_GBK[27019] := 16#C24D;
   // UNICODE_TO_GBK[27020] := 16#7FF9;
   // UNICODE_TO_GBK[27021] := 16#C24E;
   // UNICODE_TO_GBK[27022] := 16#7FFA;
   // UNICODE_TO_GBK[27023] := 16#C24F;
   // UNICODE_TO_GBK[27024] := 16#7FFB;
   // UNICODE_TO_GBK[27025] := 16#B7AD;
   // UNICODE_TO_GBK[27026] := 16#7FFC;
   // UNICODE_TO_GBK[27027] := 16#D2ED;
   // UNICODE_TO_GBK[27028] := 16#7FFD;
   // UNICODE_TO_GBK[27029] := 16#C250;
   // UNICODE_TO_GBK[27030] := 16#7FFE;
   // UNICODE_TO_GBK[27031] := 16#C251;
   // UNICODE_TO_GBK[27032] := 16#7FFF;
   // UNICODE_TO_GBK[27033] := 16#C252;
   // UNICODE_TO_GBK[27034] := 16#8000;
   // UNICODE_TO_GBK[27035] := 16#D2AB;
   // UNICODE_TO_GBK[27036] := 16#8001;
   // UNICODE_TO_GBK[27037] := 16#C0CF;
   // UNICODE_TO_GBK[27038] := 16#8002;
   // UNICODE_TO_GBK[27039] := 16#C253;
   // UNICODE_TO_GBK[27040] := 16#8003;
   // UNICODE_TO_GBK[27041] := 16#BFBC;
   // UNICODE_TO_GBK[27042] := 16#8004;
   // UNICODE_TO_GBK[27043] := 16#EBA3;
   // UNICODE_TO_GBK[27044] := 16#8005;
   // UNICODE_TO_GBK[27045] := 16#D5DF;
   // UNICODE_TO_GBK[27046] := 16#8006;
   // UNICODE_TO_GBK[27047] := 16#EAC8;
   // UNICODE_TO_GBK[27048] := 16#8007;
   // UNICODE_TO_GBK[27049] := 16#C254;
   // UNICODE_TO_GBK[27050] := 16#8008;
   // UNICODE_TO_GBK[27051] := 16#C255;
   // UNICODE_TO_GBK[27052] := 16#8009;
   // UNICODE_TO_GBK[27053] := 16#C256;
   // UNICODE_TO_GBK[27054] := 16#800A;
   // UNICODE_TO_GBK[27055] := 16#C257;
   // UNICODE_TO_GBK[27056] := 16#800B;
   // UNICODE_TO_GBK[27057] := 16#F1F3;
   // UNICODE_TO_GBK[27058] := 16#800C;
   // UNICODE_TO_GBK[27059] := 16#B6F8;
   // UNICODE_TO_GBK[27060] := 16#800D;
   // UNICODE_TO_GBK[27061] := 16#CBA3;
   // UNICODE_TO_GBK[27062] := 16#800E;
   // UNICODE_TO_GBK[27063] := 16#C258;
   // UNICODE_TO_GBK[27064] := 16#800F;
   // UNICODE_TO_GBK[27065] := 16#C259;
   // UNICODE_TO_GBK[27066] := 16#8010;
   // UNICODE_TO_GBK[27067] := 16#C4CD;
   // UNICODE_TO_GBK[27068] := 16#8011;
   // UNICODE_TO_GBK[27069] := 16#C25A;
   // UNICODE_TO_GBK[27070] := 16#8012;
   // UNICODE_TO_GBK[27071] := 16#F1E7;
   // UNICODE_TO_GBK[27072] := 16#8013;
   // UNICODE_TO_GBK[27073] := 16#C25B;
   // UNICODE_TO_GBK[27074] := 16#8014;
   // UNICODE_TO_GBK[27075] := 16#F1E8;
   // UNICODE_TO_GBK[27076] := 16#8015;
   // UNICODE_TO_GBK[27077] := 16#B8FB;
   // UNICODE_TO_GBK[27078] := 16#8016;
   // UNICODE_TO_GBK[27079] := 16#F1E9;
   // UNICODE_TO_GBK[27080] := 16#8017;
   // UNICODE_TO_GBK[27081] := 16#BAC4;
   // UNICODE_TO_GBK[27082] := 16#8018;
   // UNICODE_TO_GBK[27083] := 16#D4C5;
   // UNICODE_TO_GBK[27084] := 16#8019;
   // UNICODE_TO_GBK[27085] := 16#B0D2;
   // UNICODE_TO_GBK[27086] := 16#801A;
   // UNICODE_TO_GBK[27087] := 16#C25C;
   // UNICODE_TO_GBK[27088] := 16#801B;
   // UNICODE_TO_GBK[27089] := 16#C25D;
   // UNICODE_TO_GBK[27090] := 16#801C;
   // UNICODE_TO_GBK[27091] := 16#F1EA;
   // UNICODE_TO_GBK[27092] := 16#801D;
   // UNICODE_TO_GBK[27093] := 16#C25E;
   // UNICODE_TO_GBK[27094] := 16#801E;
   // UNICODE_TO_GBK[27095] := 16#C25F;
   // UNICODE_TO_GBK[27096] := 16#801F;
   // UNICODE_TO_GBK[27097] := 16#C260;
   // UNICODE_TO_GBK[27098] := 16#8020;
   // UNICODE_TO_GBK[27099] := 16#F1EB;
   // UNICODE_TO_GBK[27100] := 16#8021;
   // UNICODE_TO_GBK[27101] := 16#C261;
   // UNICODE_TO_GBK[27102] := 16#8022;
   // UNICODE_TO_GBK[27103] := 16#F1EC;
   // UNICODE_TO_GBK[27104] := 16#8023;
   // UNICODE_TO_GBK[27105] := 16#C262;
   // UNICODE_TO_GBK[27106] := 16#8024;
   // UNICODE_TO_GBK[27107] := 16#C263;
   // UNICODE_TO_GBK[27108] := 16#8025;
   // UNICODE_TO_GBK[27109] := 16#F1ED;
   // UNICODE_TO_GBK[27110] := 16#8026;
   // UNICODE_TO_GBK[27111] := 16#F1EE;
   // UNICODE_TO_GBK[27112] := 16#8027;
   // UNICODE_TO_GBK[27113] := 16#F1EF;
   // UNICODE_TO_GBK[27114] := 16#8028;
   // UNICODE_TO_GBK[27115] := 16#F1F1;
   // UNICODE_TO_GBK[27116] := 16#8029;
   // UNICODE_TO_GBK[27117] := 16#F1F0;
   // UNICODE_TO_GBK[27118] := 16#802A;
   // UNICODE_TO_GBK[27119] := 16#C5D5;
   // UNICODE_TO_GBK[27120] := 16#802B;
   // UNICODE_TO_GBK[27121] := 16#C264;
   // UNICODE_TO_GBK[27122] := 16#802C;
   // UNICODE_TO_GBK[27123] := 16#C265;
   // UNICODE_TO_GBK[27124] := 16#802D;
   // UNICODE_TO_GBK[27125] := 16#C266;
   // UNICODE_TO_GBK[27126] := 16#802E;
   // UNICODE_TO_GBK[27127] := 16#C267;
   // UNICODE_TO_GBK[27128] := 16#802F;
   // UNICODE_TO_GBK[27129] := 16#C268;
   // UNICODE_TO_GBK[27130] := 16#8030;
   // UNICODE_TO_GBK[27131] := 16#C269;
   // UNICODE_TO_GBK[27132] := 16#8031;
   // UNICODE_TO_GBK[27133] := 16#F1F2;
   // UNICODE_TO_GBK[27134] := 16#8032;
   // UNICODE_TO_GBK[27135] := 16#C26A;
   // UNICODE_TO_GBK[27136] := 16#8033;
   // UNICODE_TO_GBK[27137] := 16#B6FA;
   // UNICODE_TO_GBK[27138] := 16#8034;
   // UNICODE_TO_GBK[27139] := 16#C26B;
   // UNICODE_TO_GBK[27140] := 16#8035;
   // UNICODE_TO_GBK[27141] := 16#F1F4;
   // UNICODE_TO_GBK[27142] := 16#8036;
   // UNICODE_TO_GBK[27143] := 16#D2AE;
   // UNICODE_TO_GBK[27144] := 16#8037;
   // UNICODE_TO_GBK[27145] := 16#DEC7;
   // UNICODE_TO_GBK[27146] := 16#8038;
   // UNICODE_TO_GBK[27147] := 16#CBCA;
   // UNICODE_TO_GBK[27148] := 16#8039;
   // UNICODE_TO_GBK[27149] := 16#C26C;
   // UNICODE_TO_GBK[27150] := 16#803A;
   // UNICODE_TO_GBK[27151] := 16#C26D;
   // UNICODE_TO_GBK[27152] := 16#803B;
   // UNICODE_TO_GBK[27153] := 16#B3DC;
   // UNICODE_TO_GBK[27154] := 16#803C;
   // UNICODE_TO_GBK[27155] := 16#C26E;
   // UNICODE_TO_GBK[27156] := 16#803D;
   // UNICODE_TO_GBK[27157] := 16#B5A2;
   // UNICODE_TO_GBK[27158] := 16#803E;
   // UNICODE_TO_GBK[27159] := 16#C26F;
   // UNICODE_TO_GBK[27160] := 16#803F;
   // UNICODE_TO_GBK[27161] := 16#B9A2;
   // UNICODE_TO_GBK[27162] := 16#8040;
   // UNICODE_TO_GBK[27163] := 16#C270;
   // UNICODE_TO_GBK[27164] := 16#8041;
   // UNICODE_TO_GBK[27165] := 16#C271;
   // UNICODE_TO_GBK[27166] := 16#8042;
   // UNICODE_TO_GBK[27167] := 16#C4F4;
   // UNICODE_TO_GBK[27168] := 16#8043;
   // UNICODE_TO_GBK[27169] := 16#F1F5;
   // UNICODE_TO_GBK[27170] := 16#8044;
   // UNICODE_TO_GBK[27171] := 16#C272;
   // UNICODE_TO_GBK[27172] := 16#8045;
   // UNICODE_TO_GBK[27173] := 16#C273;
   // UNICODE_TO_GBK[27174] := 16#8046;
   // UNICODE_TO_GBK[27175] := 16#F1F6;
   // UNICODE_TO_GBK[27176] := 16#8047;
   // UNICODE_TO_GBK[27177] := 16#C274;
   // UNICODE_TO_GBK[27178] := 16#8048;
   // UNICODE_TO_GBK[27179] := 16#C275;
   // UNICODE_TO_GBK[27180] := 16#8049;
   // UNICODE_TO_GBK[27181] := 16#C276;
   // UNICODE_TO_GBK[27182] := 16#804A;
   // UNICODE_TO_GBK[27183] := 16#C1C4;
   // UNICODE_TO_GBK[27184] := 16#804B;
   // UNICODE_TO_GBK[27185] := 16#C1FB;
   // UNICODE_TO_GBK[27186] := 16#804C;
   // UNICODE_TO_GBK[27187] := 16#D6B0;
   // UNICODE_TO_GBK[27188] := 16#804D;
   // UNICODE_TO_GBK[27189] := 16#F1F7;
   // UNICODE_TO_GBK[27190] := 16#804E;
   // UNICODE_TO_GBK[27191] := 16#C277;
   // UNICODE_TO_GBK[27192] := 16#804F;
   // UNICODE_TO_GBK[27193] := 16#C278;
   // UNICODE_TO_GBK[27194] := 16#8050;
   // UNICODE_TO_GBK[27195] := 16#C279;
   // UNICODE_TO_GBK[27196] := 16#8051;
   // UNICODE_TO_GBK[27197] := 16#C27A;
   // UNICODE_TO_GBK[27198] := 16#8052;
   // UNICODE_TO_GBK[27199] := 16#F1F8;
   // UNICODE_TO_GBK[27200] := 16#8053;
   // UNICODE_TO_GBK[27201] := 16#C27B;
   // UNICODE_TO_GBK[27202] := 16#8054;
   // UNICODE_TO_GBK[27203] := 16#C1AA;
   // UNICODE_TO_GBK[27204] := 16#8055;
   // UNICODE_TO_GBK[27205] := 16#C27C;
   // UNICODE_TO_GBK[27206] := 16#8056;
   // UNICODE_TO_GBK[27207] := 16#C27D;
   // UNICODE_TO_GBK[27208] := 16#8057;
   // UNICODE_TO_GBK[27209] := 16#C27E;
   // UNICODE_TO_GBK[27210] := 16#8058;
   // UNICODE_TO_GBK[27211] := 16#C6B8;
   // UNICODE_TO_GBK[27212] := 16#8059;
   // UNICODE_TO_GBK[27213] := 16#C280;
   // UNICODE_TO_GBK[27214] := 16#805A;
   // UNICODE_TO_GBK[27215] := 16#BEDB;
   // UNICODE_TO_GBK[27216] := 16#805B;
   // UNICODE_TO_GBK[27217] := 16#C281;
   // UNICODE_TO_GBK[27218] := 16#805C;
   // UNICODE_TO_GBK[27219] := 16#C282;
   // UNICODE_TO_GBK[27220] := 16#805D;
   // UNICODE_TO_GBK[27221] := 16#C283;
   // UNICODE_TO_GBK[27222] := 16#805E;
   // UNICODE_TO_GBK[27223] := 16#C284;
   // UNICODE_TO_GBK[27224] := 16#805F;
   // UNICODE_TO_GBK[27225] := 16#C285;
   // UNICODE_TO_GBK[27226] := 16#8060;
   // UNICODE_TO_GBK[27227] := 16#C286;
   // UNICODE_TO_GBK[27228] := 16#8061;
   // UNICODE_TO_GBK[27229] := 16#C287;
   // UNICODE_TO_GBK[27230] := 16#8062;
   // UNICODE_TO_GBK[27231] := 16#C288;
   // UNICODE_TO_GBK[27232] := 16#8063;
   // UNICODE_TO_GBK[27233] := 16#C289;
   // UNICODE_TO_GBK[27234] := 16#8064;
   // UNICODE_TO_GBK[27235] := 16#C28A;
   // UNICODE_TO_GBK[27236] := 16#8065;
   // UNICODE_TO_GBK[27237] := 16#C28B;
   // UNICODE_TO_GBK[27238] := 16#8066;
   // UNICODE_TO_GBK[27239] := 16#C28C;
   // UNICODE_TO_GBK[27240] := 16#8067;
   // UNICODE_TO_GBK[27241] := 16#C28D;
   // UNICODE_TO_GBK[27242] := 16#8068;
   // UNICODE_TO_GBK[27243] := 16#C28E;
   // UNICODE_TO_GBK[27244] := 16#8069;
   // UNICODE_TO_GBK[27245] := 16#F1F9;
   // UNICODE_TO_GBK[27246] := 16#806A;
   // UNICODE_TO_GBK[27247] := 16#B4CF;
   // UNICODE_TO_GBK[27248] := 16#806B;
   // UNICODE_TO_GBK[27249] := 16#C28F;
   // UNICODE_TO_GBK[27250] := 16#806C;
   // UNICODE_TO_GBK[27251] := 16#C290;
   // UNICODE_TO_GBK[27252] := 16#806D;
   // UNICODE_TO_GBK[27253] := 16#C291;
   // UNICODE_TO_GBK[27254] := 16#806E;
   // UNICODE_TO_GBK[27255] := 16#C292;
   // UNICODE_TO_GBK[27256] := 16#806F;
   // UNICODE_TO_GBK[27257] := 16#C293;
   // UNICODE_TO_GBK[27258] := 16#8070;
   // UNICODE_TO_GBK[27259] := 16#C294;
   // UNICODE_TO_GBK[27260] := 16#8071;
   // UNICODE_TO_GBK[27261] := 16#F1FA;
   // UNICODE_TO_GBK[27262] := 16#8072;
   // UNICODE_TO_GBK[27263] := 16#C295;
   // UNICODE_TO_GBK[27264] := 16#8073;
   // UNICODE_TO_GBK[27265] := 16#C296;
   // UNICODE_TO_GBK[27266] := 16#8074;
   // UNICODE_TO_GBK[27267] := 16#C297;
   // UNICODE_TO_GBK[27268] := 16#8075;
   // UNICODE_TO_GBK[27269] := 16#C298;
   // UNICODE_TO_GBK[27270] := 16#8076;
   // UNICODE_TO_GBK[27271] := 16#C299;
   // UNICODE_TO_GBK[27272] := 16#8077;
   // UNICODE_TO_GBK[27273] := 16#C29A;
   // UNICODE_TO_GBK[27274] := 16#8078;
   // UNICODE_TO_GBK[27275] := 16#C29B;
   // UNICODE_TO_GBK[27276] := 16#8079;
   // UNICODE_TO_GBK[27277] := 16#C29C;
   // UNICODE_TO_GBK[27278] := 16#807A;
   // UNICODE_TO_GBK[27279] := 16#C29D;
   // UNICODE_TO_GBK[27280] := 16#807B;
   // UNICODE_TO_GBK[27281] := 16#C29E;
   // UNICODE_TO_GBK[27282] := 16#807C;
   // UNICODE_TO_GBK[27283] := 16#C29F;
   // UNICODE_TO_GBK[27284] := 16#807D;
   // UNICODE_TO_GBK[27285] := 16#C2A0;
   // UNICODE_TO_GBK[27286] := 16#807E;
   // UNICODE_TO_GBK[27287] := 16#C340;
   // UNICODE_TO_GBK[27288] := 16#807F;
   // UNICODE_TO_GBK[27289] := 16#EDB2;
   // UNICODE_TO_GBK[27290] := 16#8080;
   // UNICODE_TO_GBK[27291] := 16#EDB1;
   // UNICODE_TO_GBK[27292] := 16#8081;
   // UNICODE_TO_GBK[27293] := 16#C341;
   // UNICODE_TO_GBK[27294] := 16#8082;
   // UNICODE_TO_GBK[27295] := 16#C342;
   // UNICODE_TO_GBK[27296] := 16#8083;
   // UNICODE_TO_GBK[27297] := 16#CBE0;
   // UNICODE_TO_GBK[27298] := 16#8084;
   // UNICODE_TO_GBK[27299] := 16#D2DE;
   // UNICODE_TO_GBK[27300] := 16#8085;
   // UNICODE_TO_GBK[27301] := 16#C343;
   // UNICODE_TO_GBK[27302] := 16#8086;
   // UNICODE_TO_GBK[27303] := 16#CBC1;
   // UNICODE_TO_GBK[27304] := 16#8087;
   // UNICODE_TO_GBK[27305] := 16#D5D8;
   // UNICODE_TO_GBK[27306] := 16#8088;
   // UNICODE_TO_GBK[27307] := 16#C344;
   // UNICODE_TO_GBK[27308] := 16#8089;
   // UNICODE_TO_GBK[27309] := 16#C8E2;
   // UNICODE_TO_GBK[27310] := 16#808A;
   // UNICODE_TO_GBK[27311] := 16#C345;
   // UNICODE_TO_GBK[27312] := 16#808B;
   // UNICODE_TO_GBK[27313] := 16#C0DF;
   // UNICODE_TO_GBK[27314] := 16#808C;
   // UNICODE_TO_GBK[27315] := 16#BCA1;
   // UNICODE_TO_GBK[27316] := 16#808D;
   // UNICODE_TO_GBK[27317] := 16#C346;
   // UNICODE_TO_GBK[27318] := 16#808E;
   // UNICODE_TO_GBK[27319] := 16#C347;
   // UNICODE_TO_GBK[27320] := 16#808F;
   // UNICODE_TO_GBK[27321] := 16#C348;
   // UNICODE_TO_GBK[27322] := 16#8090;
   // UNICODE_TO_GBK[27323] := 16#C349;
   // UNICODE_TO_GBK[27324] := 16#8091;
   // UNICODE_TO_GBK[27325] := 16#C34A;
